ACTION ResetLockDepalletizing_2_action:
LockDepalletizing := FALSE;
END_ACTION

ACTION Check_StackIn__entry:
Delay.IN:=FALSE;
Delay();
END_ACTION

ACTION Check_StackIn__action:
Delay.IN:=ST08_404_B52_2.BitInToCheck;
Delay.PT:=T#3500ms;
Delay();
END_ACTION

ACTION VakuumOff_action:
ST08_403_Y50_6.MoveInit := TRUE;
ST08_403_Y50_7.MoveInit := TRUE;
END_ACTION

ACTION VakuumOff__action:
ST08_403_Y50_6.MoveInit := TRUE;
ST08_403_Y50_7.MoveInit := TRUE;
END_ACTION

ACTION SetLockDepalletizing_3_action:
LockDepalletizing := TRUE;
END_ACTION

ACTION CheckFixerPal_1_entry:
ProcessMessage02:='2IM1';(*'Abstapler wartet auf Aufstapler*)
END_ACTION

ACTION CheckFixerPal_1_exit:
ProcessMessage02:='';
END_ACTION

ACTION UnLocking_Trays_1__action:
ST08_405_Y53_4.MoveWork:=TRUE;
END_ACTION

ACTION Depallatizing_Unlock8_action:
LockDepalletizing := FALSE;
END_ACTION

ACTION Wait_Tray_entry:
Delay.IN:=FALSE;
Delay();
Timeout();
ProcessMessage01:='';
END_ACTION

ACTION Wait_Tray_action:
Delay(IN:=	NOT ST08_402_B51_2.BitInToCheck AND
     		ST08_404_B52_2.BitInToCheck
    ,PT:=T#300ms);

(*Damit der Aufstapler weitermachen kann, wenn kein Blister mehr kommt*)
Timeout(IN:=	NOT Delay.Q AND ST08_Palletizing.State=STATE_RUN, PT:=T#15s);
ProcessMessage01:='1IM16';(*ST. 8 warte aut Tray in HV vor Schleuse einlauf*)
END_ACTION

ACTION Locking_Trays___entry:
Timeout(IN:=FALSE);
END_ACTION

ACTION Locking_Trays___action:
ST08_405_Y53_4.MoveInit:=TRUE;
END_ACTION

ACTION Locking_Trays___exit:
gNewStackIn:=FALSE;
END_ACTION

ACTION Check_Blister__entry:
Delay(IN:=FALSE);
Timeout(IN:=FALSE);
END_ACTION

ACTION Check_Blister__action:
Delay(IN:=ST08_404_B52_3.BitInToCheck ,PT:=T#3000ms);
END_ACTION

ACTION Msg_SpecialMenu_entry:
MessageHandler.ClearMessageLines(sVisu:=Visu.Message);

MsgID:='PM200';
MsgString:='Blister falsche Lage in Blistereinlauf';
MsgString:=CONCAT(MsgString,'$R$N');
MsgString:=CONCAT(MsgString,'Lage korrigieren und weiter mit OK');
END_ACTION

ACTION Msg_SpecialMenu_action:
MessageHandler.Msg.ID:=MsgID;
MessageHandler.Msg.Name:='St8_Stop';
MessageHandler.Msg.Text:=MsgString;
MessageHandler.Msg.Color:=Color.red;
MessageHandler.Msg.Station:=5;
MessageHandler.MsgButton1Text:='continue';

MessageHandler(
	Prio:=2, 							(*1=highest, .. , 4=lowest*)
	Btn1Addr:=ADR(MsgOk),			(*Address of Button1 , if Zero then Button is unvisible*)
	Btn2Addr:=0,	(*Address of Button2 , if Zero then Button is unvisible*)
	sVisu:=Visu.Message);

MessageHandler.DisableMultiSelect(sVisu:=Visu.Message);
END_ACTION

ACTION Msg_SpecialMenu_exit:
MsgOk:=FALSE;
MsgCancel:=FALSE;
MessageHandler.ClearMessageLines(sVisu:=Visu.Message);
END_ACTION

ACTION Wait_DoorClose12_entry:
ProcessMessage01:='';
END_ACTION

ACTION Wait_DoorClose12_action:
ProcessMessage01:='1IM17';(*St. 8 warte Türe 2 Einlauf geschlossen*)
END_ACTION

ACTION Wait_DoorClose12_exit:
ProcessMessage01:='';
END_ACTION

ACTION Belt_on_action:
ConveyorOn:=TRUE;
END_ACTION

ACTION VRZ_open_action:
ST08_402_Y50_4.MoveWork:=TRUE;
END_ACTION

ACTION schieben_work_action:
ST08_402_Y52_7.MoveWork:=TRUE;
END_ACTION

ACTION Blister_Out_entry:
ProcessMessage01:='';
END_ACTION

ACTION Blister_Out_action:
ProcessMessage01:='1IM18';(*St. 8 warte aut Tray in Schleuse einlauf*)
END_ACTION

ACTION Blister_Out_exit:
gNewStackIn:=TRUE;
gRequestNewStack:=FALSE;
END_ACTION

ACTION VRZ_close_action:
ST08_402_Y50_4.MoveInit:=TRUE;
END_ACTION

ACTION schieben_init_action:
ST08_402_Y52_7.MoveInit:=TRUE;
END_ACTION

ACTION Belt_off_action:
ConveyorOn:=FALSE;
END_ACTION

ACTION Settling_time__entry:
Delay.IN:=FALSE;
Delay();
END_ACTION

ACTION Settling_time__action:
Delay.IN:=TRUE;
Delay.PT:=t#1000ms;
Delay();
END_ACTION

ACTION Check_StackIn___entry:
gRequestNewStack:=TRUE;
END_ACTION

ACTION Wait_DoorClose4_entry:
ProcessMessage01:='';
END_ACTION

ACTION Wait_DoorClose4_action:
ProcessMessage01:='1IM19';(*St.8 warte Türe 1 einlauf geschlossen*)
END_ACTION

ACTION Wait_DoorClose4_exit:
ProcessMessage01:='';
END_ACTION

ACTION Door_open_13_action:
ST08_405_Y51_0.MoveWork:=TRUE;
END_ACTION

ACTION VRZ_open_13_action:
ST08_404_Y51_6.MoveWork:=TRUE;
END_ACTION

ACTION Belt_on_13_action:
ConveyorOn:=TRUE;
END_ACTION

ACTION Check_TrayIn___entry:
ProcessMessage01:='';
END_ACTION

ACTION Check_TrayIn___action:
ProcessMessage01:='1IM20';(*St.4 warte auf Tray in Reinigungsposition*)
END_ACTION

ACTION Check_TrayIn___exit:
ProcessMessage01:='';
END_ACTION

ACTION VRZ_close_12_action:
ST08_404_Y51_6.MoveInit:=TRUE;
END_ACTION

ACTION Door_CLOSE_12_action:
ST08_405_Y51_0.MoveInit:=TRUE;
END_ACTION

ACTION Wait_DoorClose_5_entry:
ProcessMessage01:='';
END_ACTION

ACTION Wait_DoorClose_5_action:
ProcessMessage01:='1IM21';(*St.8 warte Türe 2 einlauf geschlossen*)
END_ACTION

ACTION Wait_DoorClose_5_exit:
ProcessMessage01:='';
END_ACTION

ACTION Belt_off_12_action:
ConveyorOn:=FALSE;
END_ACTION

ACTION ResultOk_action:
Result:=RESULT_OK;
END_ACTION

ACTION eWaitLastTray_entry:
ProcessMessage02:='EMPTY';
END_ACTION

ACTION eWaitLastTray_action:
ProcessMessage02:='2IM7';(*Aufstapler leerfahren*)
END_ACTION

ACTION eWaitLastTray_exit:
ProcessMessage02:='2IM8';(*Halb vollen Blister rausfahren*)
END_ACTION

ACTION eSetLockDepalletizing_2_action:
LockDepalletizing := TRUE;
END_ACTION

ACTION eM_Abstapeln_mitte_entry:
ST08_180_M1.MoveAbs:=TRUE;
ST08_180_M1.Vorgabe_Pos_Abs:=TD.PosAbstapeln[2].Pos;	(*1=unten, 2= mitte, 3=oben, 4=frei*)
END_ACTION

ACTION eLifter_Short_up_action:
ST08_404_Y53_0.MoveWork:=TRUE;
END_ACTION

ACTION eLifter_Long_down_action:
ST08_404_Y53_2.MoveInit:=TRUE;
END_ACTION

ACTION eVakuumOn_action:
ST08_403_Y50_6.MoveWork := TRUE;
ST08_403_Y50_7.MoveWork := TRUE;
END_ACTION

ACTION eCheckFixerPal__entry:
ProcessMessage02:='2IM1';(*'Abstapler wartet auf Aufstapler*)
END_ACTION

ACTION eCheckFixerPal__exit:
ProcessMessage02:='';
END_ACTION

ACTION eUnLocking_Trays__action:
ST08_405_Y53_4.MoveWork:=TRUE;
END_ACTION

ACTION eM_Abstapeln_unten___entry:
ST08_180_M1.MoveAbs:=TRUE;
ST08_180_M1.Vorgabe_Pos_Abs:=TD.PosAbstapeln[1].Pos;	(*1=unten, 2= mitte, 3=oben, 4=frei*)
END_ACTION

ACTION eLifter_Short_Down__action:
ST08_404_Y53_0.MoveInit:=TRUE;
END_ACTION

ACTION eResetLockDepalletizing_3_action:
LockDepalletizing := FALSE;
END_ACTION

ACTION eVakuumOff_action:
ST08_403_Y50_6.MoveInit := TRUE;
ST08_403_Y50_7.MoveInit := TRUE;
END_ACTION

ACTION eMsgEndRunEmpty_entry:
MessageHandler.ClearMessageLines(sVisu:=Visu.Message);
MsgOk:=FALSE;
ProcessMessage02:='EMPTY';
END_ACTION

ACTION eMsgEndRunEmpty_action:
MessageHandler.Msg.ID:='PM21';
MessageHandler.Msg.Name:='Maschine ist leergefahren';
MessageHandler.Msg.Text:= 'Maschine ist leergefahren';
MessageHandler.Msg.Color:=	Color.yellow ;
MessageHandler.Msg.Station:=1;

MessageHandler(
	Prio:=2, 					(*1=highest, .. , 4=lowest*)
	Btn1Addr:=ADR(MsgOk),		(*Address of Button1 , if Zero then Button is unvisible*)
	Btn2Addr:=0,				(*Address of Button2 , if Zero then Button is unvisible*)
	sVisu:=Visu.Message);

IF ModeSelect.Mode<=MODE_MANUAL THEN
	MsgOk:=TRUE;
END_IF
END_ACTION

ACTION eMsgEndRunEmpty_exit:
MsgOk:=FALSE;
ModeSelect.AskForManual:=TRUE;
gRunEmpty:=FALSE;
END_ACTION

ACTION SeqEnd_action:
SFCTime:=TIME_TO_DINT(TIME()-SFCTimeStart);
State:=STATE_WAIT;
END_ACTION

TRANSITION StateOk:
ST08_405_Y51_0.State=STATE_OK
END_TRANSITION

TRANSITION OK:
ST00_226_S2.BitInToCheck=FALSE
END_TRANSITION

TRANSITION with_Motor:
MP.ST08.StapelMotor
END_TRANSITION

TRANSITION MotorOn:
ST08_180_M1.On
END_TRANSITION

TRANSITION busy:
ST08_180_M1.Busy
END_TRANSITION

TRANSITION Done:
ST08_180_M1.Done
END_TRANSITION

TRANSITION StateOk:
ST08_404_Y53_2.State=STATE_OK
END_TRANSITION

TRANSITION StateOk:
ST08_404_Y53_0.State=STATE_OK
END_TRANSITION

TRANSITION OLD_:
NOT gNewStackIn AND
ST08_405_Y53_4.InitPosition
END_TRANSITION

TRANSITION free:
NOT ST08_Palletizing.LockPalletizing
END_TRANSITION

TRANSITION CheckClosePal:
ST08_408_B56_1.ValveSensor AND	 	(* Rückhaltezylinder links Auslauf STN8 GST *)
ST08_408_B56_3.ValveSensor 			(* Rückhaltezylinder rechts Auslauf STN8 GST *)
END_TRANSITION

TRANSITION StateOk:
ST08_405_Y53_4.State=STATE_OK
END_TRANSITION

TRANSITION with_Motor:
MP.ST08.StapelMotor
END_TRANSITION

TRANSITION on:
ST08_180_M1.on
END_TRANSITION

TRANSITION busy:
ST08_180_M1.Busy
END_TRANSITION

TRANSITION Done:
ST08_180_M1.Done
END_TRANSITION

TRANSITION StateOk:
ST08_404_Y53_0.State=STATE_OK
END_TRANSITION

TRANSITION StateOk:
ST08_405_Y53_4.State=STATE_OK
END_TRANSITION

TRANSITION with_Motor:
MP.ST08.StapelMotor
END_TRANSITION

TRANSITION VacuumOn:
ST08_403_Y50_6.State=STATE_OK AND
ST08_403_Y50_7.State=STATE_OK
END_TRANSITION

TRANSITION on:
ST08_180_M1.on
END_TRANSITION

TRANSITION busy:
ST08_180_M1.Busy
END_TRANSITION

TRANSITION Done:
ST08_180_M1.Done
END_TRANSITION

TRANSITION StateOk:
ST08_404_Y53_0.State=STATE_OK
END_TRANSITION

TRANSITION OK:
ST08_404_B52_2.BitInToCheck=FALSE OR Delay.Q
END_TRANSITION

TRANSITION VacuumOff:
ST08_403_Y50_6.State=STATE_OK AND
ST08_403_Y50_7.State=STATE_OK
END_TRANSITION

TRANSITION OK:
  DelayOut.Q
END_TRANSITION

TRANSITION Empty_:
Delay.Q
END_TRANSITION

TRANSITION free:
NOT ST08_Palletizing.LockPalletizing
END_TRANSITION

TRANSITION AutoStop:
		ModeSelect.Mode=MODE_AUTO_STOP
OR	ModeSelect.Mode=MODE_STEP_STOP
END_TRANSITION

TRANSITION with_Motor:
MP.ST08.StapelMotor
END_TRANSITION

TRANSITION MotorOn:
ST08_180_M1.On
END_TRANSITION

TRANSITION busy:
ST08_180_M1.Busy
END_TRANSITION

TRANSITION Done:
ST08_180_M1.Done
END_TRANSITION

TRANSITION StateOk:
ST08_404_Y53_0.State=STATE_OK
END_TRANSITION

TRANSITION StateOk:
ST08_404_Y53_2.State=STATE_OK
END_TRANSITION

TRANSITION VakuumOn:
ST08_403_Y50_6.State=STATE_OK AND
ST08_403_Y50_7.State=STATE_OK
END_TRANSITION

TRANSITION CheckClosePal:
ST08_408_B56_1.ValveSensor AND	 	(* Rückhaltezylinder links Auslauf STN8 GST *)
ST08_408_B56_3.ValveSensor 			(* Rückhaltezylinder rechts Auslauf STN8 GST *)
END_TRANSITION

TRANSITION StateOk:
ST08_405_Y53_4.State=STATE_OK
END_TRANSITION

TRANSITION with_Motor:
MP.ST08.StapelMotor
END_TRANSITION

TRANSITION MotorOn:
ST08_180_M1.On
END_TRANSITION

TRANSITION busy:
ST08_180_M1.Busy
END_TRANSITION

TRANSITION Done:
ST08_180_M1.Done
END_TRANSITION

TRANSITION StateOk:
ST08_404_Y53_2.State=STATE_OK
END_TRANSITION

TRANSITION StateOk:
ST08_405_Y53_4.State=STATE_OK
END_TRANSITION

TRANSITION with_Motor:
MP.ST08.StapelMotor
END_TRANSITION

TRANSITION MotorOn:
ST08_180_M1.On
END_TRANSITION

TRANSITION busy:
ST08_180_M1.Busy
END_TRANSITION

TRANSITION Done:
ST08_180_M1.Done
END_TRANSITION

TRANSITION StateOk:
ST08_404_Y53_0.State=STATE_OK
END_TRANSITION

TRANSITION In_:
ST08_404_B52_2.BitInToCheck=FALSE
END_TRANSITION

TRANSITION VakuumOff:
ST08_403_Y50_6.State=STATE_OK AND
ST08_403_Y50_7.State=STATE_OK
END_TRANSITION

TRANSITION Empty__:
Delay.Q
END_TRANSITION

TRANSITION VakuumOff:
ST08_403_Y50_6.State=STATE_OK AND
ST08_403_Y50_7.State=STATE_OK
END_TRANSITION

TRANSITION Trans90:
NOT ST08_Palletizing.LockPalletizing
END_TRANSITION

TRANSITION CheckClosePal:
ST08_408_B56_1.ValveSensor AND	 	(* Rückhaltezylinder links Auslauf STN8 GST *)
ST08_408_B56_3.ValveSensor 			(* Rückhaltezylinder rechts Auslauf STN8 GST *)
END_TRANSITION

TRANSITION StateOk:
ST08_405_Y53_4.State=STATE_OK
END_TRANSITION

TRANSITION AutoStop:
		ModeSelect.Mode=MODE_AUTO_STOP
OR	ModeSelect.Mode=MODE_STEP_STOP
END_TRANSITION

TRANSITION StateOk:
ST08_405_Y53_4.State=STATE_OK
END_TRANSITION

TRANSITION OK:
ST08_404_B52_3.BitInToCheck=FALSE OR
MP.ST03.SGM_3621
END_TRANSITION

TRANSITION TimeOut:
Delay.Q
END_TRANSITION

TRANSITION MsgOk:
		ST08_404_B52_3.BitInToCheck=FALSE
OR	MsgOk
END_TRANSITION

TRANSITION OK:
ST00_226_S2.BitInToCheck=FALSE
END_TRANSITION

TRANSITION StateOk:
ST08_402_Y50_4.State=STATE_OK
END_TRANSITION

TRANSITION mit_schieben:
MP.ST08.Traystapel_schieben
END_TRANSITION

TRANSITION #StateOk:
ST08_402_Y52_7.State=STATE_OK
END_TRANSITION

TRANSITION WTOut:
ST08_404_B52_2.BitInToCheck=FALSE AND ST08_402_B51_2.BitInToCheck=TRUE
END_TRANSITION

TRANSITION StateOk:
ST08_402_Y50_4.State=STATE_OK
END_TRANSITION

TRANSITION mit_schieben:
MP.ST08.Traystapel_schieben
END_TRANSITION

TRANSITION StateOk:
ST08_402_Y52_7.State=STATE_OK
END_TRANSITION

TRANSITION OK:
ST08_402_B51_5.BitInToCheck
END_TRANSITION

TRANSITION IN__:
 ST08_404_B52_2.BitInToCheck=FALSE
END_TRANSITION

TRANSITION OK:
NOT ST00_226_S1.BitInToCheck AND
NOT ST00_229_S1.BitInToCheck
END_TRANSITION

TRANSITION StateOk:
ST08_405_Y51_0.State=STATE_OK AND
ST08_404_Y51_6.State=STATE_OK
END_TRANSITION

TRANSITION OK:
    ST08_406_B54_0.BitInToCheck=FALSE AND ST08_404_B52_2.BitInToCheck=TRUE
END_TRANSITION

TRANSITION StateOk:
ST08_404_Y51_6.State=STATE_OK AND
ST08_405_Y51_0.State=STATE_OK
END_TRANSITION

TRANSITION OK:
ST00_226_S2.BitInToCheck=FALSE
END_TRANSITION

TRANSITION wait:
ST08_Palletizing.WaitLastTray
END_TRANSITION

TRANSITION voll:
NOT ST08_404_B52_2.BitInToCheck 		(*Traystapel in Ablageposition Isokörper*)
END_TRANSITION

TRANSITION leer:
ST08_404_B52_2.BitInToCheck 		(*Traystapel in Ablageposition Isokörper*)
END_TRANSITION

TRANSITION free:
NOT ST08_Palletizing.LockPalletizing
END_TRANSITION

TRANSITION with_Motor:
MP.ST08.StapelMotor
END_TRANSITION

TRANSITION MotorOn:
ST08_180_M1.On
END_TRANSITION

TRANSITION busy:
ST08_180_M1.Busy
END_TRANSITION

TRANSITION Done:
ST08_180_M1.Done
END_TRANSITION

TRANSITION StateOk:
ST08_404_Y53_0.State=STATE_OK
END_TRANSITION

TRANSITION StateOk:
ST08_404_Y53_2.State=STATE_OK
END_TRANSITION

TRANSITION VakuumOn:
ST08_403_Y50_6.State=STATE_OK AND
ST08_403_Y50_7.State=STATE_OK
END_TRANSITION

TRANSITION CheckClosePal:
ST08_408_B56_1.ValveSensor AND	 	(* Rückhaltezylinder links Auslauf STN8 GST *)
ST08_408_B56_3.ValveSensor 			(* Rückhaltezylinder rechts Auslauf STN8 GST *)
END_TRANSITION

TRANSITION StateOk:
ST08_405_Y53_4.State=STATE_OK
END_TRANSITION

TRANSITION with_Motor:
MP.ST08.StapelMotor
END_TRANSITION

TRANSITION MotorOn:
ST08_180_M1.On
END_TRANSITION

TRANSITION busy:
ST08_180_M1.Busy
END_TRANSITION

TRANSITION Done:
ST08_180_M1.Done
END_TRANSITION

TRANSITION StateOk:
ST08_404_Y53_0.State=STATE_OK
END_TRANSITION

TRANSITION VakuumOff:
ST08_403_Y50_6.State=STATE_OK AND
ST08_403_Y50_7.State=STATE_OK
END_TRANSITION

TRANSITION wait:
ST08_Palletizing.State = STATE_WAIT
END_TRANSITION
END_PROGRAM

(* POU Stations/ST_00/ST00_SFCs/_SpecialModeSFCs/SpecialMode01, SFC *)
PROGRAM SpecialMode01 (*Feeding-Test: Pickup Part with Robot01 from Feeder and put it into NOK-Box *)
(* Date: 07.DEZ 2010    Author: Ext/g.baiz  *)

VAR_OUTPUT
	SFCCurrentPOU		: STRING:='SpecialMode01';
	SFCCurrentStep	: STRING:='';
	SFCTime					:	DINT;
  State   				:	DINT;
  Result  				:	DINT;
END_VAR
VAR_INPUT
	Start						:	BOOL;
END_VAR
VAR
	MsgOK				:	BOOL;
	MsgCancel		:	BOOL;
	SFCRun					:	BOOL;
	SFCTimeStart		:	TIME;
	(* Userdefinded area *)



END_VAR
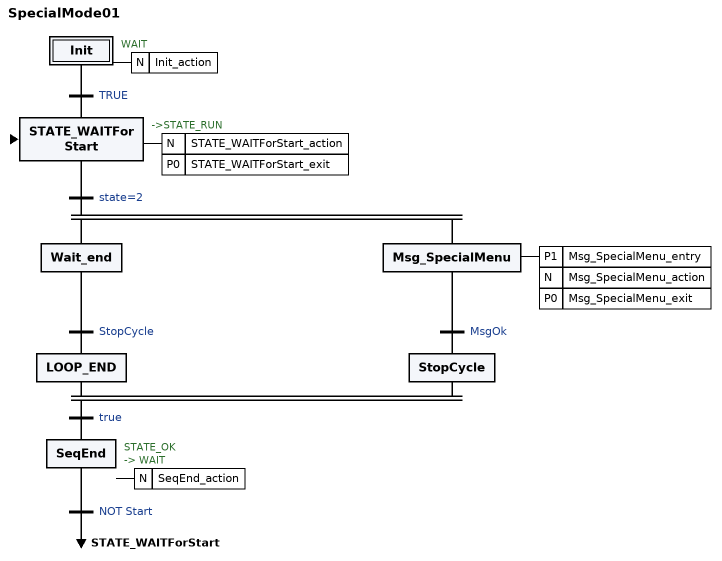
INITIAL_STEP Init: (* WAIT *)
	Init_action(N);
END_STEP
TRANSITION FROM Init TO STATE_WAITForStart := TRUE;
END_TRANSITION
STEP STATE_WAITForStart: (* ->STATE_RUN *)
	STATE_WAITForStart_action(N);
	STATE_WAITForStart_exit(P0);
END_STEP
TRANSITION FROM STATE_WAITForStart TO (Wait_end, Msg_SpecialMenu) := state=2;
END_TRANSITION
STEP Wait_end:
END_STEP
TRANSITION FROM Wait_end TO LOOP_END := StopCycle;
END_TRANSITION
STEP LOOP_END:
END_STEP
STEP Msg_SpecialMenu:
	Msg_SpecialMenu_entry(P1);
	Msg_SpecialMenu_action(N);
	Msg_SpecialMenu_exit(P0);
END_STEP
TRANSITION FROM Msg_SpecialMenu TO StopCycle := MsgOk;
END_TRANSITION
STEP StopCycle:
END_STEP
TRANSITION FROM (LOOP_END, StopCycle) TO SeqEnd := true;
END_TRANSITION
STEP SeqEnd: (* STATE_OK / -> WAIT *)
	SeqEnd_action(N);
END_STEP
TRANSITION FROM SeqEnd TO STATE_WAITForStart := NOT Start;
END_TRANSITION

ACTION Init_action:
Start:=FALSE;
State:=STATE_WAIT;
END_ACTION

ACTION STATE_WAITForStart_action:
IF 	Start THEN
	State:=STATE_RUN;
	Result:=RESULT_NON;
	SFCTimeStart:=TIME();
END_IF
END_ACTION

ACTION STATE_WAITForStart_exit:
StopCycle:=FALSE;
END_ACTION

ACTION Msg_SpecialMenu_entry:
MessageHandler.ClearMessageLines(sVisu:=Visu.Message);
StopCycle:=FALSE;
END_ACTION

ACTION Msg_SpecialMenu_action:
MessageHandler.Msg.ID:='PM50';
MessageHandler.Msg.Name:='SP1_Stop';
MessageHandler.Msg.Text:='Teilablauf beenden mit <OK>';
MessageHandler.Msg.Color:=Color.blue;
MessageHandler.Msg.Station:=0;


MessageHandler(
	Prio:=2, 									(*1=highest, .. , 4=lowest*)
	Btn1Addr:=ADR(MsgOk),			(*Address of Button1 , if Zero then Button is unvisible*)
	Btn2Addr:=0,	(*Address of Button2 , if Zero then Button is unvisible*)
	sVisu:=Visu.Message);

MessageHandler.DisableMultiSelect(sVisu:=Visu.Message);
END_ACTION

ACTION Msg_SpecialMenu_exit:
MsgOk:=FALSE;
MsgCancel:=FALSE;
StopCycle:=TRUE;
END_ACTION

ACTION SeqEnd_action:
IF 	State=STATE_RUN THEN
	SFCTime:=TIME_TO_DINT(TIME()-SFCTimeStart);
	State:=STATE_OK;
END_IF


IF 	NOT Start THEN
	State:=STATE_WAIT;
END_IF
END_ACTION
END_PROGRAM

(* POU Stations/ST_08_Palettierer/ST_08_SFCs/ST08_Palletizing, SFC *)
PROGRAM ST08_Palletizing

VAR_OUTPUT
	SFCCurrentPOU			: STRING:='ST08_Palletizing';
	SFCCurrentStep			: STRING:='';
	FB_CurrentStepHistorie	: FB_CurrentStepHistorie;
	SFCTime					: DINT;
	State   				: StateObject	:= STATE_WAIT;
	Result  				: StateResult;
	MoveInStopper			: BOOL;
END_VAR
VAR_INPUT
	TestpartMoveOut		: BOOL;
	MoveOut				: BOOL;
	ConveyorOn			: BOOL;
	LastTray			: BOOL;			(*Leerfahren. Der letzte, halbvollen Blisters ist rausgefahren*)
END_VAR
VAR
	MsgOK				: BOOL;
	MsgCancel			: BOOL;
	SFCRun				: BOOL;
	SFCTimeStart		: TIME;
	Delay				: TON;
	Error				: ErrorStruct;
	(* Userdefinded area *)
	ExitPosRdy_T		: TON;
	BlisterStart		: BOOL;
	LockInlett			:BOOL;

	WaitLastTray		:BOOL;		(*Leerfahren. Startet das Rausfahren des halbvollen Blisters*)
	LockPalletizing		:BOOL;
END_VAR
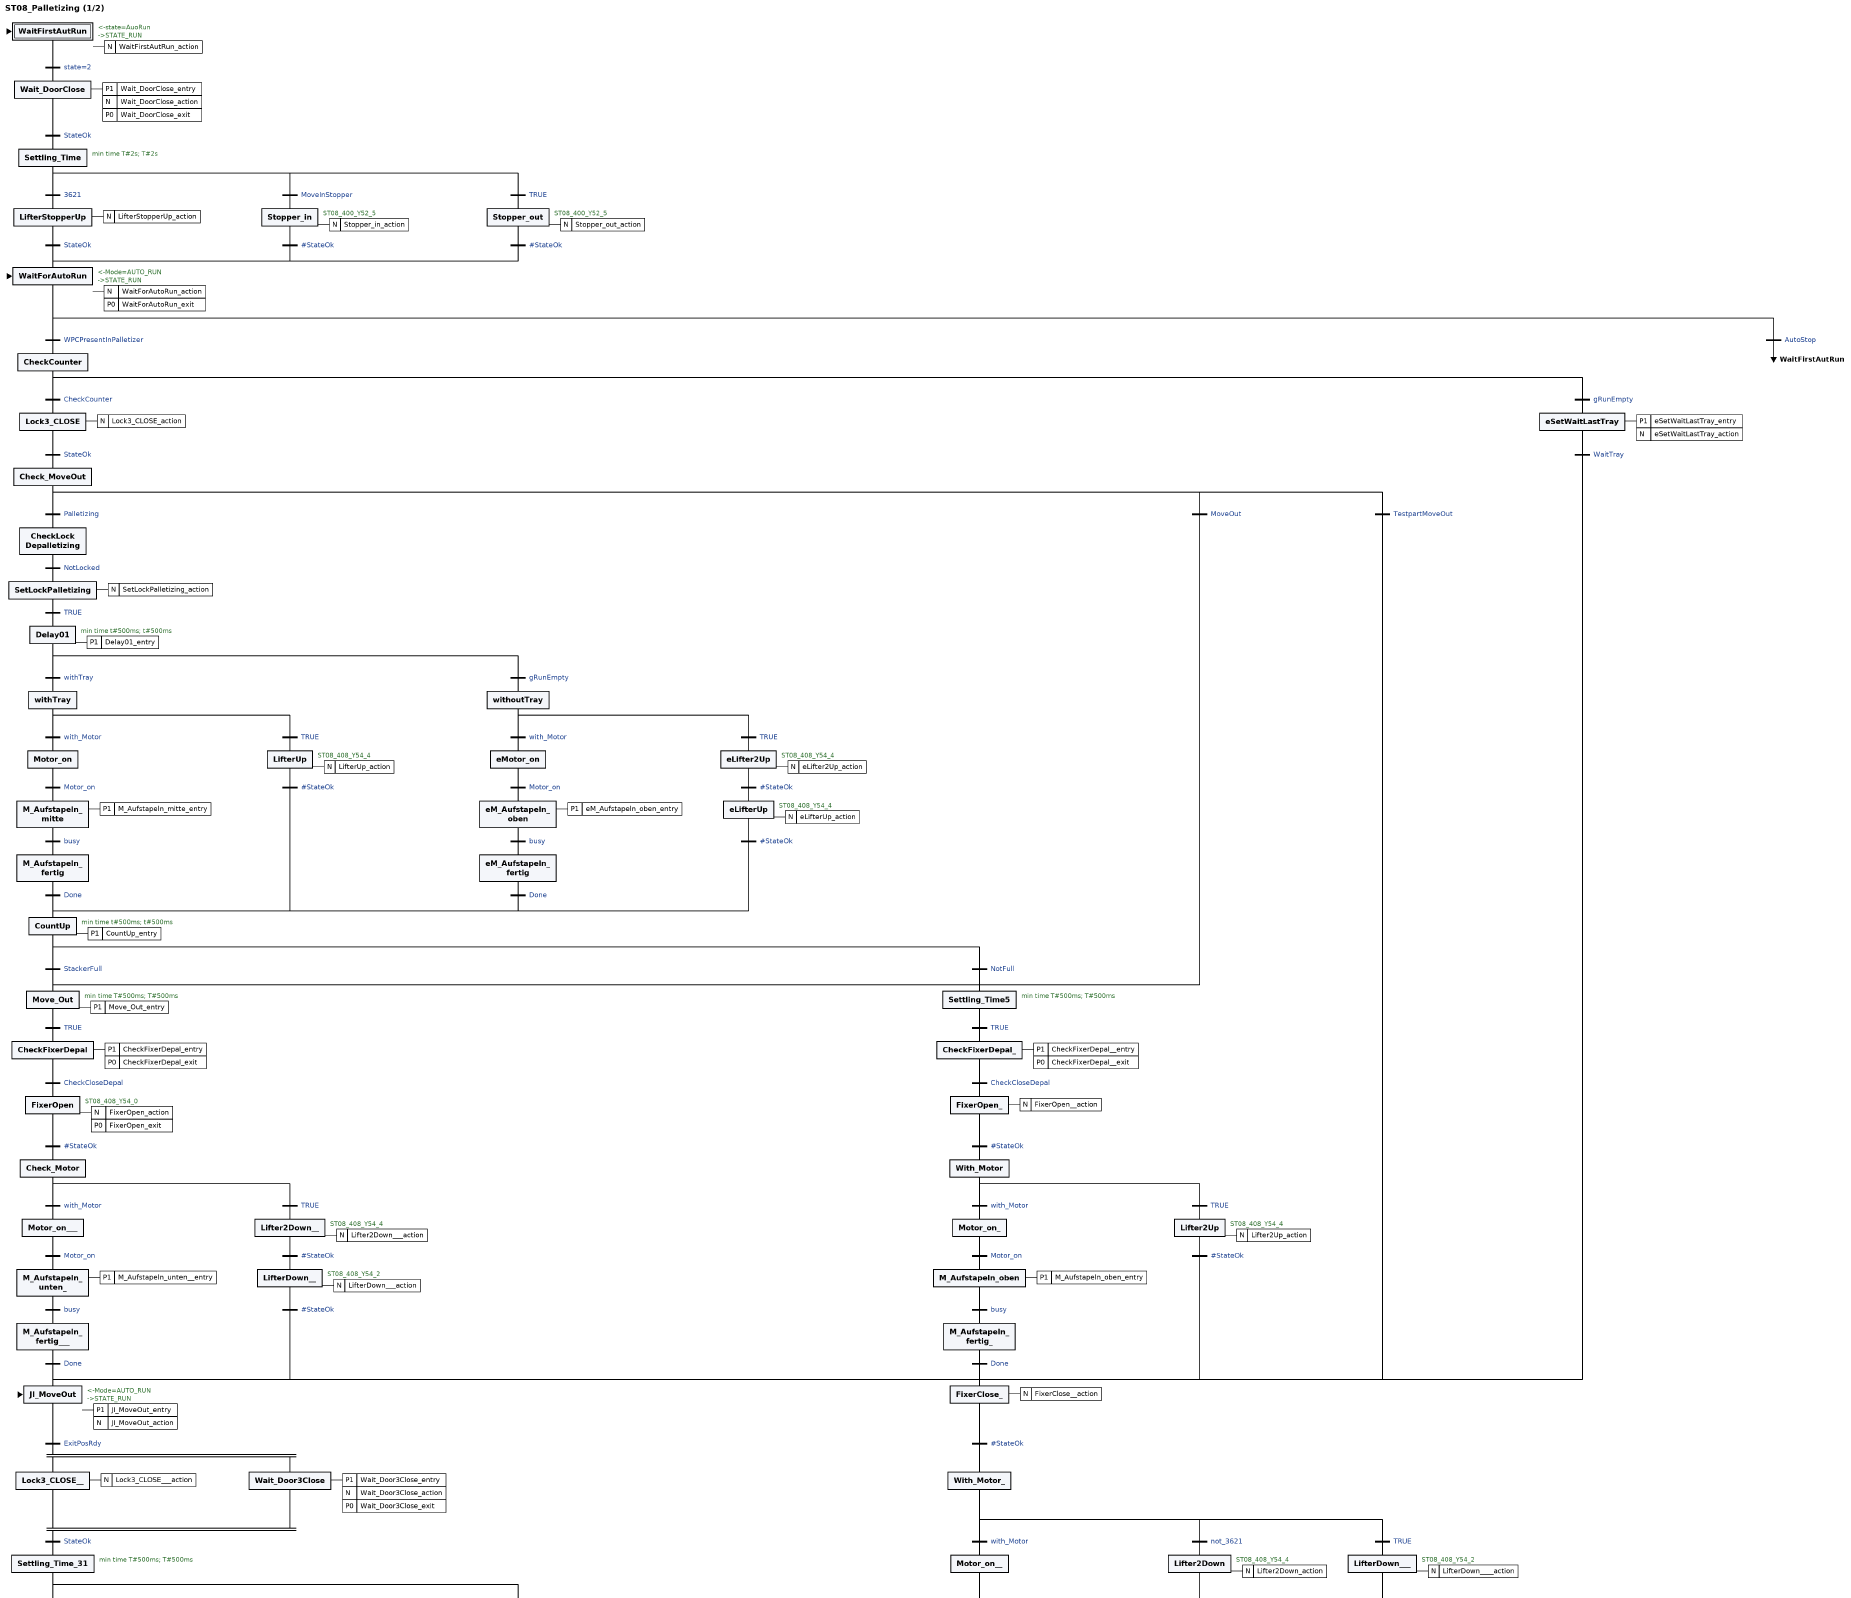
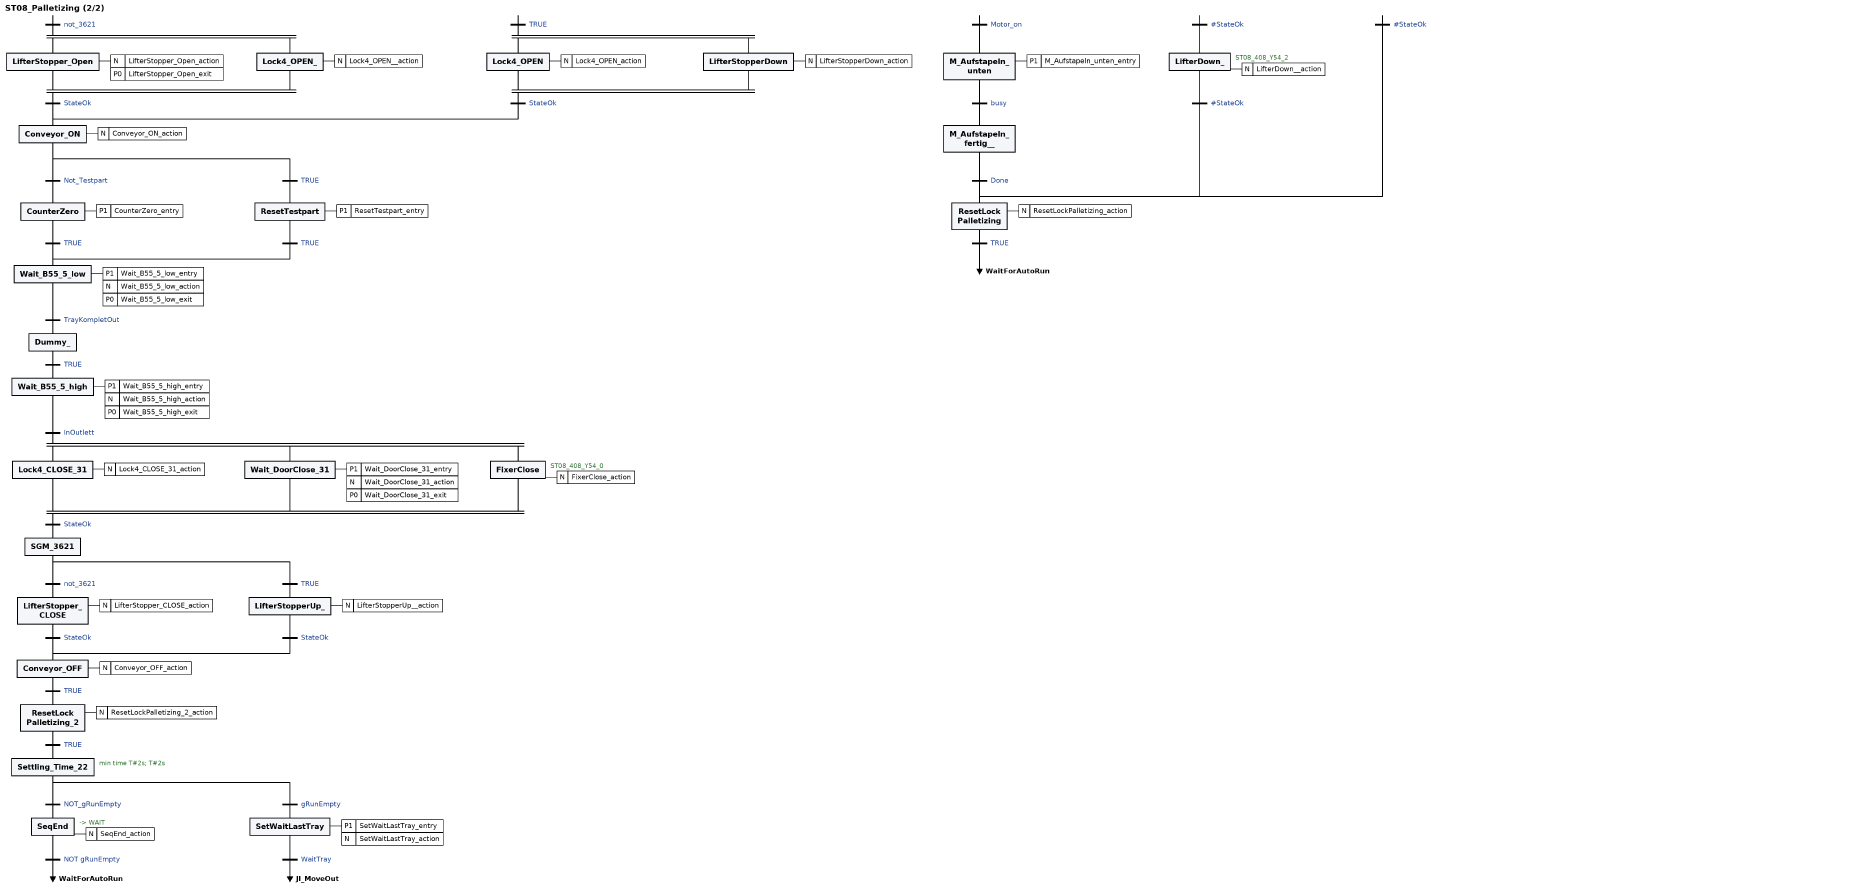
INITIAL_STEP WaitFirstAutRun: (* <-state=AuoRun / ->STATE_RUN *)
	WaitFirstAutRun_action(N);
END_STEP
TRANSITION FROM WaitFirstAutRun TO Wait_DoorClose := state=2;
END_TRANSITION
STEP Wait_DoorClose:
	Wait_DoorClose_entry(P1);
	Wait_DoorClose_action(N);
	Wait_DoorClose_exit(P0);
END_STEP
TRANSITION FROM Wait_DoorClose TO Settling_Time := StateOk;
END_TRANSITION
STEP Settling_Time: (* min time T#2s; T#2s *)
END_STEP
TRANSITION FROM Settling_Time TO LifterStopperUp := 3621;
END_TRANSITION
TRANSITION FROM Settling_Time TO Stopper_in := MoveInStopper;
END_TRANSITION
TRANSITION FROM Settling_Time TO Stopper_out := TRUE;
END_TRANSITION
STEP LifterStopperUp:
	LifterStopperUp_action(N);
END_STEP
TRANSITION FROM LifterStopperUp TO WaitForAutoRun := StateOk;
END_TRANSITION
STEP Stopper_in: (* ST08_400_Y52_5 *)
	Stopper_in_action(N);
END_STEP
TRANSITION FROM Stopper_in TO WaitForAutoRun := #StateOk;
END_TRANSITION
STEP Stopper_out: (* ST08_400_Y52_5 *)
	Stopper_out_action(N);
END_STEP
TRANSITION FROM Stopper_out TO WaitForAutoRun := #StateOk;
END_TRANSITION
STEP WaitForAutoRun: (* <-Mode=AUTO_RUN / ->STATE_RUN *)
	WaitForAutoRun_action(N);
	WaitForAutoRun_exit(P0);
END_STEP
TRANSITION FROM WaitForAutoRun TO CheckCounter := WPCPresentInPalletizer;
END_TRANSITION
TRANSITION FROM WaitForAutoRun TO WaitFirstAutRun := AutoStop;
END_TRANSITION
STEP CheckCounter:
END_STEP
TRANSITION FROM CheckCounter TO Lock3_CLOSE := CheckCounter;
END_TRANSITION
TRANSITION FROM CheckCounter TO eSetWaitLastTray := gRunEmpty;
END_TRANSITION
STEP eSetWaitLastTray:
	eSetWaitLastTray_entry(P1);
	eSetWaitLastTray_action(N);
END_STEP
TRANSITION FROM eSetWaitLastTray TO JI_MoveOut := WaitTray;
END_TRANSITION
STEP Lock3_CLOSE:
	Lock3_CLOSE_action(N);
END_STEP
TRANSITION FROM Lock3_CLOSE TO Check_MoveOut := StateOk;
END_TRANSITION
STEP Check_MoveOut:
END_STEP
TRANSITION FROM Check_MoveOut TO CheckLockDepalletizing := Palletizing;
END_TRANSITION
TRANSITION FROM Check_MoveOut TO Move_Out := MoveOut;
END_TRANSITION
TRANSITION FROM Check_MoveOut TO JI_MoveOut := TestpartMoveOut;
END_TRANSITION
STEP CheckLockDepalletizing:
END_STEP
TRANSITION FROM CheckLockDepalletizing TO SetLockPalletizing := NotLocked;
END_TRANSITION
STEP SetLockPalletizing:
	SetLockPalletizing_action(N);
END_STEP
TRANSITION FROM SetLockPalletizing TO Delay01 := TRUE;
END_TRANSITION
STEP Delay01: (* min time t#500ms; t#500ms *)
	Delay01_entry(P1);
END_STEP
TRANSITION FROM Delay01 TO withTray := withTray;
END_TRANSITION
TRANSITION FROM Delay01 TO withoutTray := gRunEmpty;
END_TRANSITION
STEP withTray:
END_STEP
TRANSITION FROM withTray TO Motor_on := with_Motor;
END_TRANSITION
TRANSITION FROM withTray TO LifterUp := TRUE;
END_TRANSITION
STEP Motor_on:
END_STEP
TRANSITION FROM Motor_on TO M_Aufstapeln_mitte := Motor_on;
END_TRANSITION
STEP M_Aufstapeln_mitte:
	M_Aufstapeln_mitte_entry(P1);
END_STEP
TRANSITION FROM M_Aufstapeln_mitte TO M_Aufstapeln_fertig := busy;
END_TRANSITION
STEP M_Aufstapeln_fertig:
END_STEP
TRANSITION FROM M_Aufstapeln_fertig TO CountUp := Done;
END_TRANSITION
STEP LifterUp: (* ST08_408_Y54_4 *)
	LifterUp_action(N);
END_STEP
TRANSITION FROM LifterUp TO CountUp := #StateOk;
END_TRANSITION
STEP withoutTray:
END_STEP
TRANSITION FROM withoutTray TO eMotor_on := with_Motor;
END_TRANSITION
TRANSITION FROM withoutTray TO eLifter2Up := TRUE;
END_TRANSITION
STEP eMotor_on:
END_STEP
TRANSITION FROM eMotor_on TO eM_Aufstapeln_oben := Motor_on;
END_TRANSITION
STEP eM_Aufstapeln_oben:
	eM_Aufstapeln_oben_entry(P1);
END_STEP
TRANSITION FROM eM_Aufstapeln_oben TO eM_Aufstapeln_fertig := busy;
END_TRANSITION
STEP eM_Aufstapeln_fertig:
END_STEP
TRANSITION FROM eM_Aufstapeln_fertig TO CountUp := Done;
END_TRANSITION
STEP eLifter2Up: (* ST08_408_Y54_4 *)
	eLifter2Up_action(N);
END_STEP
TRANSITION FROM eLifter2Up TO eLifterUp := #StateOk;
END_TRANSITION
STEP eLifterUp: (* ST08_408_Y54_4 *)
	eLifterUp_action(N);
END_STEP
TRANSITION FROM eLifterUp TO CountUp := #StateOk;
END_TRANSITION
STEP CountUp: (* min time t#500ms; t#500ms *)
	CountUp_entry(P1);
END_STEP
TRANSITION FROM CountUp TO Move_Out := StackerFull;
END_TRANSITION
TRANSITION FROM CountUp TO Settling_Time5 := NotFull;
END_TRANSITION
STEP Settling_Time5: (* min time T#500ms; T#500ms *)
END_STEP
TRANSITION FROM Settling_Time5 TO CheckFixerDepal_ := TRUE;
END_TRANSITION
STEP CheckFixerDepal_:
	CheckFixerDepal__entry(P1);
	CheckFixerDepal__exit(P0);
END_STEP
TRANSITION FROM CheckFixerDepal_ TO FixerOpen_ := CheckCloseDepal;
END_TRANSITION
STEP FixerOpen_:
	FixerOpen__action(N);
END_STEP
TRANSITION FROM FixerOpen_ TO With_Motor := #StateOk;
END_TRANSITION
STEP With_Motor:
END_STEP
TRANSITION FROM With_Motor TO Motor_on_ := with_Motor;
END_TRANSITION
TRANSITION FROM With_Motor TO Lifter2Up := TRUE;
END_TRANSITION
STEP Motor_on_:
END_STEP
TRANSITION FROM Motor_on_ TO M_Aufstapeln_oben := Motor_on;
END_TRANSITION
STEP M_Aufstapeln_oben:
	M_Aufstapeln_oben_entry(P1);
END_STEP
TRANSITION FROM M_Aufstapeln_oben TO M_Aufstapeln_fertig_ := busy;
END_TRANSITION
STEP M_Aufstapeln_fertig_:
END_STEP
TRANSITION FROM M_Aufstapeln_fertig_ TO FixerClose_ := Done;
END_TRANSITION
STEP Lifter2Up: (* ST08_408_Y54_4 *)
	Lifter2Up_action(N);
END_STEP
TRANSITION FROM Lifter2Up TO FixerClose_ := #StateOk;
END_TRANSITION
STEP FixerClose_:
	FixerClose__action(N);
END_STEP
TRANSITION FROM FixerClose_ TO With_Motor_ := #StateOk;
END_TRANSITION
STEP With_Motor_:
END_STEP
TRANSITION FROM With_Motor_ TO Motor_on__ := with_Motor;
END_TRANSITION
TRANSITION FROM With_Motor_ TO Lifter2Down := not_3621;
END_TRANSITION
TRANSITION FROM With_Motor_ TO LifterDown___ := TRUE;
END_TRANSITION
STEP Motor_on__:
END_STEP
TRANSITION FROM Motor_on__ TO M_Aufstapeln_unten := Motor_on;
END_TRANSITION
STEP M_Aufstapeln_unten:
	M_Aufstapeln_unten_entry(P1);
END_STEP
TRANSITION FROM M_Aufstapeln_unten TO M_Aufstapeln_fertig__ := busy;
END_TRANSITION
STEP M_Aufstapeln_fertig__:
END_STEP
TRANSITION FROM M_Aufstapeln_fertig__ TO ResetLockPalletizing := Done;
END_TRANSITION
STEP Lifter2Down: (* ST08_408_Y54_4 *)
	Lifter2Down_action(N);
END_STEP
TRANSITION FROM Lifter2Down TO LifterDown_ := #StateOk;
END_TRANSITION
STEP LifterDown_: (* ST08_408_Y54_2 *)
	LifterDown__action(N);
END_STEP
TRANSITION FROM LifterDown_ TO ResetLockPalletizing := #StateOk;
END_TRANSITION
STEP LifterDown___: (* ST08_408_Y54_2 *)
	LifterDown____action(N);
END_STEP
TRANSITION FROM LifterDown___ TO ResetLockPalletizing := #StateOk;
END_TRANSITION
STEP ResetLockPalletizing:
	ResetLockPalletizing_action(N);
END_STEP
TRANSITION FROM ResetLockPalletizing TO WaitForAutoRun := TRUE;
END_TRANSITION
STEP Move_Out: (* min time T#500ms; T#500ms *)
	Move_Out_entry(P1);
END_STEP
TRANSITION FROM Move_Out TO CheckFixerDepal := TRUE;
END_TRANSITION
STEP CheckFixerDepal:
	CheckFixerDepal_entry(P1);
	CheckFixerDepal_exit(P0);
END_STEP
TRANSITION FROM CheckFixerDepal TO FixerOpen := CheckCloseDepal;
END_TRANSITION
STEP FixerOpen: (* ST08_408_Y54_0 *)
	FixerOpen_action(N);
	FixerOpen_exit(P0);
END_STEP
TRANSITION FROM FixerOpen TO Check_Motor := #StateOk;
END_TRANSITION
STEP Check_Motor:
END_STEP
TRANSITION FROM Check_Motor TO Motor_on___ := with_Motor;
END_TRANSITION
TRANSITION FROM Check_Motor TO Lifter2Down__ := TRUE;
END_TRANSITION
STEP Motor_on___:
END_STEP
TRANSITION FROM Motor_on___ TO M_Aufstapeln_unten_ := Motor_on;
END_TRANSITION
STEP M_Aufstapeln_unten_:
	M_Aufstapeln_unten__entry(P1);
END_STEP
TRANSITION FROM M_Aufstapeln_unten_ TO M_Aufstapeln_fertig___ := busy;
END_TRANSITION
STEP M_Aufstapeln_fertig___:
END_STEP
TRANSITION FROM M_Aufstapeln_fertig___ TO JI_MoveOut := Done;
END_TRANSITION
STEP Lifter2Down__: (* ST08_408_Y54_4 *)
	Lifter2Down___action(N);
END_STEP
TRANSITION FROM Lifter2Down__ TO LifterDown__ := #StateOk;
END_TRANSITION
STEP LifterDown__: (* ST08_408_Y54_2 *)
	LifterDown___action(N);
END_STEP
TRANSITION FROM LifterDown__ TO JI_MoveOut := #StateOk;
END_TRANSITION
STEP JI_MoveOut: (* <-Mode=AUTO_RUN / ->STATE_RUN *)
	JI_MoveOut_entry(P1);
	JI_MoveOut_action(N);
END_STEP
TRANSITION FROM JI_MoveOut TO (Lock3_CLOSE__, Wait_Door3Close) := ExitPosRdy;
END_TRANSITION
STEP Lock3_CLOSE__:
	Lock3_CLOSE___action(N);
END_STEP
STEP Wait_Door3Close:
	Wait_Door3Close_entry(P1);
	Wait_Door3Close_action(N);
	Wait_Door3Close_exit(P0);
END_STEP
TRANSITION FROM (Lock3_CLOSE__, Wait_Door3Close) TO Settling_Time_31 := StateOk;
END_TRANSITION
STEP Settling_Time_31: (* min time T#500ms; T#500ms *)
END_STEP
TRANSITION FROM Settling_Time_31 TO (LifterStopper_Open, Lock4_OPEN_) := not_3621;
END_TRANSITION
TRANSITION FROM Settling_Time_31 TO (Lock4_OPEN, LifterStopperDown) := TRUE;
END_TRANSITION
STEP LifterStopper_Open:
	LifterStopper_Open_action(N);
	LifterStopper_Open_exit(P0);
END_STEP
STEP Lock4_OPEN_:
	Lock4_OPEN__action(N);
END_STEP
TRANSITION FROM (LifterStopper_Open, Lock4_OPEN_) TO Conveyor_ON := StateOk;
END_TRANSITION
STEP Lock4_OPEN:
	Lock4_OPEN_action(N);
END_STEP
STEP LifterStopperDown:
	LifterStopperDown_action(N);
END_STEP
TRANSITION FROM (Lock4_OPEN, LifterStopperDown) TO Conveyor_ON := StateOk;
END_TRANSITION
STEP Conveyor_ON:
	Conveyor_ON_action(N);
END_STEP
TRANSITION FROM Conveyor_ON TO CounterZero := Not_Testpart;
END_TRANSITION
TRANSITION FROM Conveyor_ON TO ResetTestpart := TRUE;
END_TRANSITION
STEP CounterZero:
	CounterZero_entry(P1);
END_STEP
TRANSITION FROM CounterZero TO Wait_B55_5_low := TRUE;
END_TRANSITION
STEP ResetTestpart:
	ResetTestpart_entry(P1);
END_STEP
TRANSITION FROM ResetTestpart TO Wait_B55_5_low := TRUE;
END_TRANSITION
STEP Wait_B55_5_low:
	Wait_B55_5_low_entry(P1);
	Wait_B55_5_low_action(N);
	Wait_B55_5_low_exit(P0);
END_STEP
TRANSITION FROM Wait_B55_5_low TO Dummy_ := TrayKompletOut;
END_TRANSITION
STEP Dummy_:
END_STEP
TRANSITION FROM Dummy_ TO Wait_B55_5_high := TRUE;
END_TRANSITION
STEP Wait_B55_5_high:
	Wait_B55_5_high_entry(P1);
	Wait_B55_5_high_action(N);
	Wait_B55_5_high_exit(P0);
END_STEP
TRANSITION FROM Wait_B55_5_high TO (Lock4_CLOSE_31, Wait_DoorClose_31, FixerClose) := InOutlett;
END_TRANSITION
STEP Lock4_CLOSE_31:
	Lock4_CLOSE_31_action(N);
END_STEP
STEP Wait_DoorClose_31:
	Wait_DoorClose_31_entry(P1);
	Wait_DoorClose_31_action(N);
	Wait_DoorClose_31_exit(P0);
END_STEP
STEP FixerClose: (* ST08_408_Y54_0 *)
	FixerClose_action(N);
END_STEP
TRANSITION FROM (Lock4_CLOSE_31, Wait_DoorClose_31, FixerClose) TO SGM_3621 := StateOk;
END_TRANSITION
STEP SGM_3621:
END_STEP
TRANSITION FROM SGM_3621 TO LifterStopper_CLOSE := not_3621;
END_TRANSITION
TRANSITION FROM SGM_3621 TO LifterStopperUp_ := TRUE;
END_TRANSITION
STEP LifterStopper_CLOSE:
	LifterStopper_CLOSE_action(N);
END_STEP
TRANSITION FROM LifterStopper_CLOSE TO Conveyor_OFF := StateOk;
END_TRANSITION
STEP LifterStopperUp_:
	LifterStopperUp__action(N);
END_STEP
TRANSITION FROM LifterStopperUp_ TO Conveyor_OFF := StateOk;
END_TRANSITION
STEP Conveyor_OFF:
	Conveyor_OFF_action(N);
END_STEP
TRANSITION FROM Conveyor_OFF TO ResetLockPalletizing_2 := TRUE;
END_TRANSITION
STEP ResetLockPalletizing_2:
	ResetLockPalletizing_2_action(N);
END_STEP
TRANSITION FROM ResetLockPalletizing_2 TO Settling_Time_22 := TRUE;
END_TRANSITION
STEP Settling_Time_22: (* min time T#2s; T#2s *)
END_STEP
TRANSITION FROM Settling_Time_22 TO SeqEnd := NOT_gRunEmpty;
END_TRANSITION
TRANSITION FROM Settling_Time_22 TO SetWaitLastTray := gRunEmpty;
END_TRANSITION
STEP SetWaitLastTray:
	SetWaitLastTray_entry(P1);
	SetWaitLastTray_action(N);
END_STEP
TRANSITION FROM SetWaitLastTray TO JI_MoveOut := WaitTray;
END_TRANSITION
STEP SeqEnd: (* -> WAIT *)
	SeqEnd_action(N);
END_STEP
TRANSITION FROM SeqEnd TO WaitForAutoRun := NOT gRunEmpty;
END_TRANSITION

ACTION WaitFirstAutRun_action:
IF 	ModeSelect.Mode=MODE_AUTO_RUN OR
	ModeSelect.Mode=MODE_STEP_RUN OR
	SpecialMode01.State=State_Run OR
 	SpecialMode06.State=State_Run THEN
	State:=STATE_RUN;
	Result:=RESULT_NON;
ELSE
	State:=STATE_WAIT;
END_IF
IF 	ModeSelect.Mode <> MODE_HOME_POS_RUN THEN
	ConveyorOn:=FALSE;
END_IF

MsgOK:=FALSE;
MsgCancel:=FALSE;
SFCRun:=FALSE;
BlisterStart:=FALSE;
LockInlett:=FALSE;
LockPalletizing:=FALSE;
MoveInStopper:=FALSE;
LastTray:=FALSE;
WaitLastTray:=FALSE;
END_ACTION

ACTION Wait_DoorClose_entry:
ProcessMessage01:='';
END_ACTION

ACTION Wait_DoorClose_action:
ProcessMessage01:='1IM8';(*St.8 warte Türe 4 auslauf geschlossen*)
ST08_407_Y51_4.MoveInit:=TRUE;
END_ACTION

ACTION Wait_DoorClose_exit:
ProcessMessage01:='';
END_ACTION

ACTION LifterStopperUp_action:
ST08_408_Y54_4.MoveWork:=TRUE;
END_ACTION

ACTION Stopper_in_action:
ST08_400_Y52_5.MoveWork :=TRUE; (* einfahren Stopper links + rechts Traystapel Auslaufband einfahren *)
END_ACTION

ACTION Stopper_out_action:
ST08_400_Y52_5.MoveInit :=TRUE; (* ausfahren Stopper links + rechts Traystapel Auslaufband einfahren *)
END_ACTION

ACTION WaitForAutoRun_action:
State:=STATE_WAIT;
LockInlett:=FALSE;
END_ACTION

ACTION WaitForAutoRun_exit:
State:=STATE_RUN;
Result:=RESULT_NON;
SFCTimeStart:=TIME();
END_ACTION

ACTION eSetWaitLastTray_entry:
LockInlett:=FALSE;
END_ACTION

ACTION eSetWaitLastTray_action:
WaitLastTray:=TRUE; (*damit wird im ST08_Process der halbvolle Blister ausgeschleust*)
END_ACTION

ACTION Lock3_CLOSE_action:
ST08_406_Y51_2.MoveInit:=TRUE;
END_ACTION

ACTION SetLockPalletizing_action:
LockPalletizing := TRUE;
END_ACTION

ACTION Delay01_entry:
LockInlett:=TRUE;
END_ACTION

ACTION M_Aufstapeln_mitte_entry:
ST08_185_M1.MoveAbs:=TRUE;
ST08_185_M1.Vorgabe_Pos_Abs:=TD.PosAufstapeln[2].Pos;	(*1=unten, 2= mitte, 3=oben, 4=frei*)
ST08_185_M1.Vorgabe_Velo:=1750;
END_ACTION

ACTION LifterUp_action:
ST08_408_Y54_2.MoveWork:=TRUE;
END_ACTION

ACTION eM_Aufstapeln_oben_entry:
ST08_185_M1.MoveAbs:=TRUE;
ST08_185_M1.Vorgabe_Pos_Abs:=TD.PosAufstapeln[3].Pos;	(*1=unten, 2= mitte, 3=oben, 4=frei*)
ST08_185_M1.Vorgabe_Velo:=1750;
END_ACTION

ACTION eLifter2Up_action:
ST08_408_Y54_4.MoveWork:=TRUE;
END_ACTION

ACTION eLifterUp_action:
ST08_408_Y54_2.MoveWork:=TRUE;
END_ACTION

ACTION CountUp_entry:
MP.ST08.NoOfBlisterInStackerOut:=MP.ST08.NoOfBlisterInStackerOut+1;
END_ACTION

ACTION CheckFixerDepal__entry:
ProcessMessage02:='2IM2';(*'Aufstapler wartet auf Abstapler*)
END_ACTION

ACTION CheckFixerDepal__exit:
ProcessMessage02:='';
END_ACTION

ACTION FixerOpen__action:
ST08_408_Y54_0.MoveWork:=TRUE;
END_ACTION

ACTION M_Aufstapeln_oben_entry:
ST08_185_M1.MoveAbs:=TRUE;
ST08_185_M1.Vorgabe_Pos_Abs:=TD.PosAufstapeln[3].Pos;	(*1=unten, 2= mitte, 3=oben, 4=frei*)
END_ACTION

ACTION Lifter2Up_action:
ST08_408_Y54_4.MoveWork:=TRUE;
END_ACTION

ACTION FixerClose__action:
ST08_408_Y54_0.MoveInit:=TRUE;
END_ACTION

ACTION M_Aufstapeln_unten_entry:
ST08_185_M1.MoveAbs:=TRUE;
ST08_185_M1.Vorgabe_Pos_Abs:=TD.PosAufstapeln[1].Pos;	(*1=unten, 2= mitte, 3=oben, 4=frei*)
END_ACTION

ACTION Lifter2Down_action:
ST08_408_Y54_4.MoveInit:=TRUE;
END_ACTION

ACTION LifterDown__action:
ST08_408_Y54_2.MoveInit:=TRUE;
END_ACTION

ACTION LifterDown____action:
ST08_408_Y54_2.MoveInit:=TRUE;
END_ACTION

ACTION ResetLockPalletizing_action:
LockPalletizing := FALSE;
END_ACTION

ACTION Move_Out_entry:
MoveOut:=TRUE;
END_ACTION

ACTION CheckFixerDepal_entry:
ProcessMessage02:='2IM2';(*'Aufstapler wartet auf Abstapler*)
END_ACTION

ACTION CheckFixerDepal_exit:
ProcessMessage02:='';
END_ACTION

ACTION FixerOpen_action:
ST08_408_Y54_0.MoveWork:=TRUE;
END_ACTION

ACTION FixerOpen_exit:
MP.ST03.WpcInStackFilled:=FALSE;
END_ACTION

ACTION M_Aufstapeln_unten__entry:
ST08_185_M1.MoveAbs:=TRUE;
ST08_185_M1.Vorgabe_Pos_Abs:=TD.PosAufstapeln[1].Pos;	(*1=unten, 2= mitte, 3=oben, 4=frei*)
END_ACTION

ACTION Lifter2Down___action:
ST08_408_Y54_4.MoveInit:=TRUE;
END_ACTION

ACTION LifterDown___action:
ST08_408_Y54_2.MoveInit:=TRUE;
END_ACTION

ACTION JI_MoveOut_entry:
ExitPosRdy_T(IN:=FALSE);
Delay.IN:=FALSE;
Delay();
END_ACTION

ACTION JI_MoveOut_action:
ExitPosRdy_T(IN:=
		(ModeSelect.Mode=MODE_AUTO_RUN	OR
		ModeSelect.Mode=MODE_STEP_RUN   OR
		ModeSelect.Mode=MODE_SPECIAL) AND
		ST08_409_B55_5.BitInToCheck , 	(* kein Stau im Auslauf *)
		PT:=T#2s);

Delay(IN:=TRUE,PT:=T#5s);

IF Delay.Q THEN
	MessageHandler.Msg.ID:='PM201';
	MessageHandler.Msg.Name:='St08 Stau im Auslauf';
	MessageHandler.Msg.Text:='Auslaufand voll!! Blister entnehmen!!';
	MessageHandler.Msg.Color:=Color.blue;
	MessageHandler.Msg.Station:=0;


	MessageHandler(
		Prio:=2, 		(*1=highest, .. , 4=lowest*)
		Btn1Addr:=0,	(*Address of Button1 , if Zero then Button is unvisible*)
		Btn2Addr:=0,	(*Address of Button2 , if Zero then Button is unvisible*)
		sVisu:=Visu.Message);


END_IF
END_ACTION

ACTION Lock3_CLOSE___action:
ST08_406_Y51_2.MoveInit:=TRUE;
END_ACTION

ACTION Wait_Door3Close_entry:
ProcessMessage01:='';
END_ACTION

ACTION Wait_Door3Close_action:
ProcessMessage01:='1IM11';(*St.8 warte Türe 3 auslauf geschlossen*)
END_ACTION

ACTION Wait_Door3Close_exit:
ProcessMessage01:='';
END_ACTION

ACTION LifterStopper_Open_action:
ST08_400_Y52_5.MoveWork :=TRUE;
END_ACTION

ACTION LifterStopper_Open_exit:
MoveInStopper:=TRUE;
END_ACTION

ACTION Lock4_OPEN__action:
ST08_407_Y51_4.MoveWork:=TRUE;
END_ACTION

ACTION Lock4_OPEN_action:
ST08_407_Y51_4.MoveWork:=TRUE;
END_ACTION

ACTION LifterStopperDown_action:
ST08_408_Y54_4.MoveInit:=TRUE;
END_ACTION

ACTION Conveyor_ON_action:
ConveyorOn:=TRUE;
END_ACTION

ACTION CounterZero_entry:
MP.ST08.NoOfBlisterInStackerOut:=0;
END_ACTION

ACTION ResetTestpart_entry:
TestpartMoveOut:=FALSE;
END_ACTION

ACTION Wait_B55_5_low_entry:
ProcessMessage01:='';
END_ACTION

ACTION Wait_B55_5_low_action:
ProcessMessage01:='1IM12';(*'St. 8 warte Tray ausgelaufen*)
END_ACTION

ACTION Wait_B55_5_low_exit:
ProcessMessage01:='';
END_ACTION

ACTION Wait_B55_5_high_entry:
ProcessMessage01:='';
END_ACTION

ACTION Wait_B55_5_high_action:
ProcessMessage01:='1IM13';(*St. 8 warte Tray auf Rollenbahn*)
END_ACTION

ACTION Wait_B55_5_high_exit:
MoveInStopper:=FALSE;
END_ACTION

ACTION Lock4_CLOSE_31_action:
ST08_407_Y51_4.MoveInit:=TRUE;
END_ACTION

ACTION Wait_DoorClose_31_entry:
ProcessMessage01:='';
END_ACTION

ACTION Wait_DoorClose_31_action:
ProcessMessage01:='1IM14';(*'St.8 warte Türe 4 auslauf geschlossen*)
END_ACTION

ACTION Wait_DoorClose_31_exit:
ProcessMessage01:='';
END_ACTION

ACTION FixerClose_action:
ST08_408_Y54_0.MoveInit:=TRUE;
END_ACTION

ACTION LifterStopper_CLOSE_action:
ST08_400_Y52_5.MoveInit:=TRUE;
END_ACTION

ACTION LifterStopperUp__action:
ST08_408_Y54_4.MoveWork:=TRUE;
END_ACTION

ACTION Conveyor_OFF_action:
ConveyorOn:=FALSE;
END_ACTION

ACTION ResetLockPalletizing_2_action:
LockPalletizing := FALSE;
END_ACTION

ACTION SetWaitLastTray_entry:
LockInlett:=FALSE;
END_ACTION

ACTION SetWaitLastTray_action:
WaitLastTray:=TRUE; (*damit wird im ST08_Process der halbvolle Blister ausgeschleust*)
END_ACTION

ACTION SeqEnd_action:
SFCTime:=TIME_TO_DINT(TIME()-SFCTimeStart);
State:=STATE_WAIT;
END_ACTION

TRANSITION StateOk:
ST08_407_Y51_4.State=STATE_OK AND
NOT ST00_227_S2.BitInToCheck AND
NOT ST00_230_S1.BitInToCheck
END_TRANSITION

TRANSITION 3621:
MP.ST03.SGM_3621
END_TRANSITION

TRANSITION StateOk:
ST08_408_Y54_4.State=STATE_OK

AND gTipImp
END_TRANSITION

TRANSITION #StateOk:
ST08_400_Y52_5.State=STATE_OK
AND gTipImp
END_TRANSITION

TRANSITION #StateOk:
ST08_400_Y52_5.State=STATE_OK
AND gTipImp
END_TRANSITION

TRANSITION WPCPresentInPalletizer:
(NOT ST08_407_B55_4.BitInToCheck OR
gRunEmpty)AND
gTipImp
END_TRANSITION

TRANSITION CheckCounter:
(gRunEmpty AND MP.ST08.NoOfBlisterInStackerOut >0) OR
NOT gRunEmpty
END_TRANSITION

TRANSITION gRunEmpty:
gRunEmpty AND MP.ST08.NoOfBlisterInStackerOut = 0
END_TRANSITION

TRANSITION WaitTray:
NOT ST08_407_B55_4.BitInToCheck AND	(* Tray in Aufstapelposition eingelaufen STN8 *)
LastTray AND	 (*damit wird im ST08_Process das ausschleusen des halbvollen Blisters bestätigt*)
gTipImp
END_TRANSITION

TRANSITION StateOk:
ST08_406_Y51_2.State=STATE_OK
END_TRANSITION

TRANSITION Palletizing:
NOT MoveOut AND
NOT TestpartMoveOut
END_TRANSITION

TRANSITION NotLocked:
NOT ST08_Depalletizing.LockDepalletizing
END_TRANSITION

TRANSITION withTray:
NOT ST08_407_B55_4.BitInToCheck (* Tray in Aufstapelposition eingelaufen STN8 *)
END_TRANSITION

TRANSITION with_Motor:
MP.ST08.StapelMotor
END_TRANSITION

TRANSITION Motor_on:
ST08_185_M1.On
END_TRANSITION

TRANSITION busy:
ST08_185_M1.Busy
END_TRANSITION

TRANSITION Done:
ST08_185_M1.Done
END_TRANSITION

TRANSITION #StateOk:
ST08_408_Y54_2.State=STATE_OK

AND gTipImp
END_TRANSITION

TRANSITION with_Motor:
MP.ST08.StapelMotor
END_TRANSITION

TRANSITION Motor_on:
ST08_185_M1.On
END_TRANSITION

TRANSITION busy:
ST08_185_M1.Busy
END_TRANSITION

TRANSITION Done:
ST08_185_M1.Done
END_TRANSITION

TRANSITION #StateOk:
ST08_408_Y54_4.State=STATE_OK

AND gTipImp
END_TRANSITION

TRANSITION #StateOk:
ST08_408_Y54_2.State=STATE_OK

AND gTipImp
END_TRANSITION

TRANSITION StackerFull:
MP.ST08.NoOfBlisterInStackerOut>=TD.NoOfPalletsPerStack OR
gRunEmpty
END_TRANSITION

TRANSITION NotFull:
TRUE
END_TRANSITION

TRANSITION CheckCloseDepal:
ST08_405_B53_3.ValveSensor AND	 	(* Rückhaltezylinder links Traystapel Isokörper GST *)
ST08_405_B53_5.ValveSensor 			(* Rückhaltezylinder rechts Traystapel Isokörper GST *)
END_TRANSITION

TRANSITION #StateOk:
ST08_408_Y54_0.State=STATE_OK

AND gTipImp
END_TRANSITION

TRANSITION with_Motor:
MP.ST08.StapelMotor
END_TRANSITION

TRANSITION Motor_on:
ST08_185_M1.On
END_TRANSITION

TRANSITION busy:
ST08_185_M1.Busy
END_TRANSITION

TRANSITION Done:
ST08_185_M1.Done AND
gTipImp
END_TRANSITION

TRANSITION #StateOk:
ST08_408_Y54_4.State=STATE_OK

AND gTipImp
END_TRANSITION

TRANSITION #StateOk:
ST08_408_Y54_0.State=STATE_OK

AND gTipImp
END_TRANSITION

TRANSITION with_Motor:
MP.ST08.StapelMotor
END_TRANSITION

TRANSITION Motor_on:
ST08_185_M1.On
END_TRANSITION

TRANSITION busy:
ST08_185_M1.Busy
END_TRANSITION

TRANSITION Done:
ST08_185_M1.Done AND
gTipImp
END_TRANSITION

TRANSITION not_3621:
NOT MP.ST03.SGM_3621
END_TRANSITION

TRANSITION #StateOk:
ST08_408_Y54_4.State=STATE_OK

AND gTipImp
END_TRANSITION

TRANSITION #StateOk:
ST08_408_Y54_2.State=STATE_OK

AND gTipImp
END_TRANSITION

TRANSITION #StateOk:
ST08_408_Y54_2.State=STATE_OK

AND gTipImp
END_TRANSITION

TRANSITION CheckCloseDepal:
ST08_405_B53_3.ValveSensor AND	 	(* Rückhaltezylinder links Traystapel Isokörper GST *)
ST08_405_B53_5.ValveSensor AND		(* Rückhaltezylinder rechts Traystapel Isokörper GST *)
gTipImp
END_TRANSITION

TRANSITION #StateOk:
ST08_408_Y54_0.State=STATE_OK

AND gTipImp
END_TRANSITION

TRANSITION with_Motor:
MP.ST08.StapelMotor
END_TRANSITION

TRANSITION Motor_on:
ST08_185_M1.On
END_TRANSITION

TRANSITION busy:
ST08_185_M1.Busy
END_TRANSITION

TRANSITION Done:
ST08_185_M1.Done AND
gTipImp
END_TRANSITION

TRANSITION #StateOk:
ST08_408_Y54_4.State=STATE_OK

AND gTipImp
END_TRANSITION

TRANSITION #StateOk:
ST08_408_Y54_2.State=STATE_OK

AND gTipImp
END_TRANSITION

TRANSITION ExitPosRdy:
ExitPosRdy_T.Q
END_TRANSITION

TRANSITION StateOk:
ST08_406_Y51_2.State=STATE_OK AND
NOT ST00_227_S1.BitInToCheck AND
gTipImp
END_TRANSITION

TRANSITION not_3621:
NOT MP.ST03.SGM_3621
END_TRANSITION

TRANSITION StateOk:
ST08_400_Y52_5.State=STATE_OK AND
ST08_407_Y51_4.State=STATE_OK AND
gTipImp
END_TRANSITION

TRANSITION StateOk:
ST08_408_Y54_4.State =STATE_OK AND
ST08_407_Y51_4.State=STATE_OK AND
gTipImp
END_TRANSITION

TRANSITION Not_Testpart:
NOT TestpartMoveOut
END_TRANSITION

TRANSITION AutoStop:
		ModeSelect.Mode=MODE_AUTO_STOP
OR	ModeSelect.Mode=MODE_STEP_STOP
END_TRANSITION

TRANSITION TrayKompletOut:
NOT ST08_409_B55_5.BitInToCheck AND
gTipImp
END_TRANSITION

TRANSITION InOutlett:
ST08_409_B55_5.BitInToCheck AND
gTipImp
END_TRANSITION

TRANSITION StateOk:
ST08_407_Y51_4.State=STATE_OK AND
NOT ST00_227_S2.BitInToCheck AND
NOT ST00_230_S1.BitInToCheck AND
ST08_408_Y54_0.State=STATE_OK AND
gTipImp
END_TRANSITION

TRANSITION not_3621:
NOT MP.ST03.SGM_3621
END_TRANSITION

TRANSITION StateOk:
(*ST08_408_Y54_4.State=STATE_OK*)

ST08_400_Y52_5.State=STATE_OK AND
gTipImp
END_TRANSITION

TRANSITION StateOk:
ST08_408_Y54_4.State=STATE_OK

AND gTipImp
END_TRANSITION

TRANSITION NOT_gRunEmpty:
NOT gRunEmpty OR
LastTray
END_TRANSITION

TRANSITION WaitTray:
NOT ST08_407_B55_4.BitInToCheck AND	(* Tray in Aufstapelposition eingelaufen STN8 *)
LastTray AND	 (*damit wird im ST08_Process das ausschleusen des halbvollen Blisters bestätigt*)
gTipImp
END_TRANSITION
END_PROGRAM

(* POU Stations/ST_08_Palettierer/ST_08_SFCs/ST08_Process, SFC *)
PROGRAM ST08_Process

VAR_OUTPUT
	SFCCurrentPOU			: STRING:='ST08_Process';
	SFCCurrentStep			: STRING:='';
	FB_CurrentStepHistorie	: FB_CurrentStepHistorie;
	SFCTime					: DINT;
	State   				: StateObject	:= STATE_WAIT;
	Result  				: StateResult;
	ConveyorHQE      	: BOOL;
	ConveyorOut       	: BOOL;
END_VAR
VAR_INPUT
	Start				: BOOL;
END_VAR
VAR
	MsgOK				: BOOL;
	MsgCancel			: BOOL;
	SFCRun				: BOOL;
	SFCTimeStart		: TIME;
	Delay				: TON;
	Delay1				: TON;
	Error				: ErrorStruct;
	(* Userdefinded area *)
	Pal_Ready     		: BOOL;


END_VAR
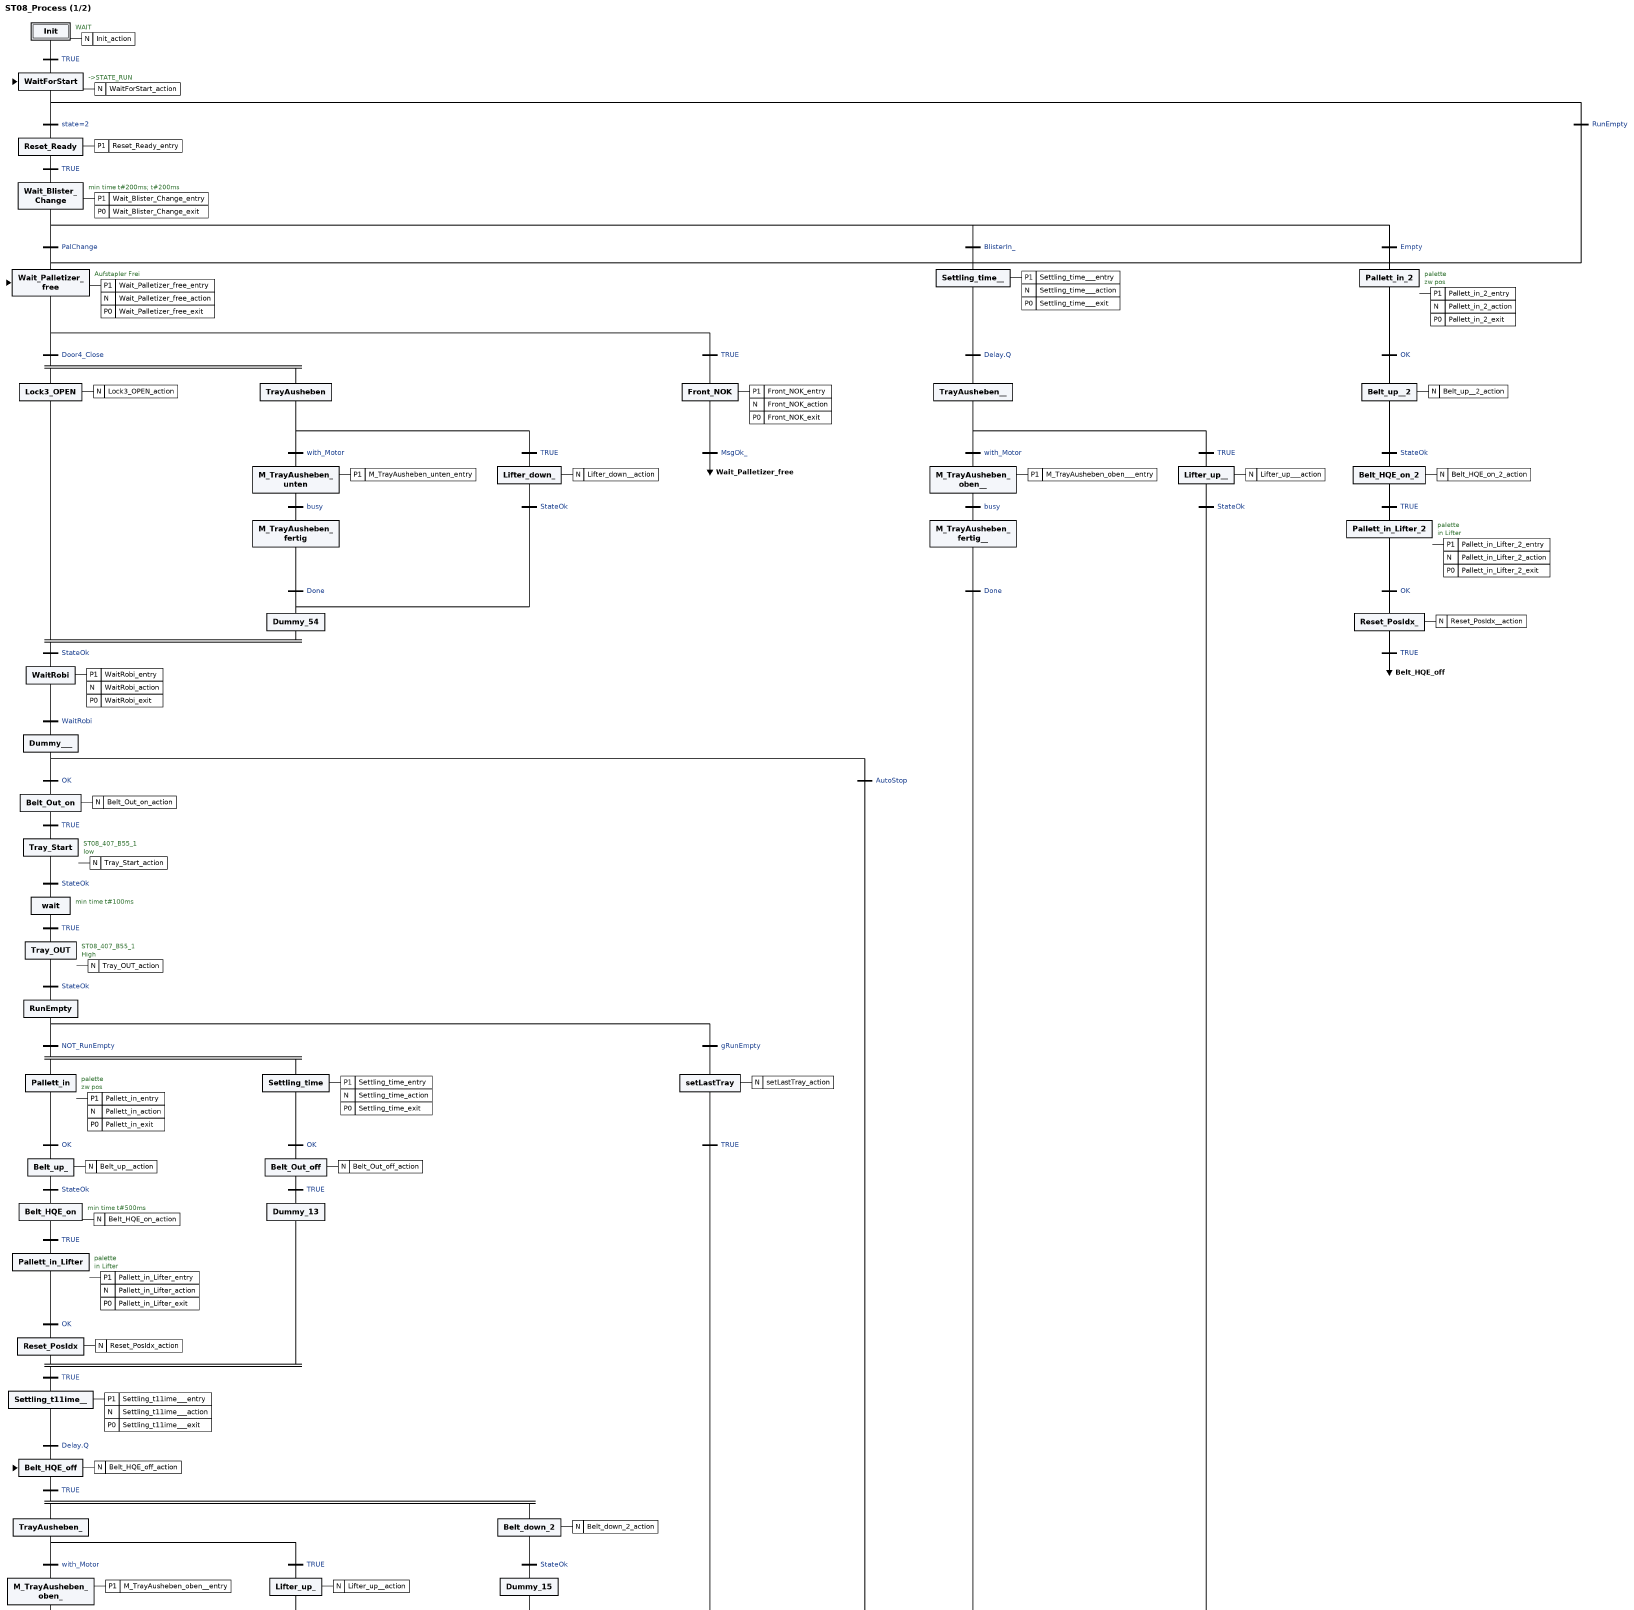
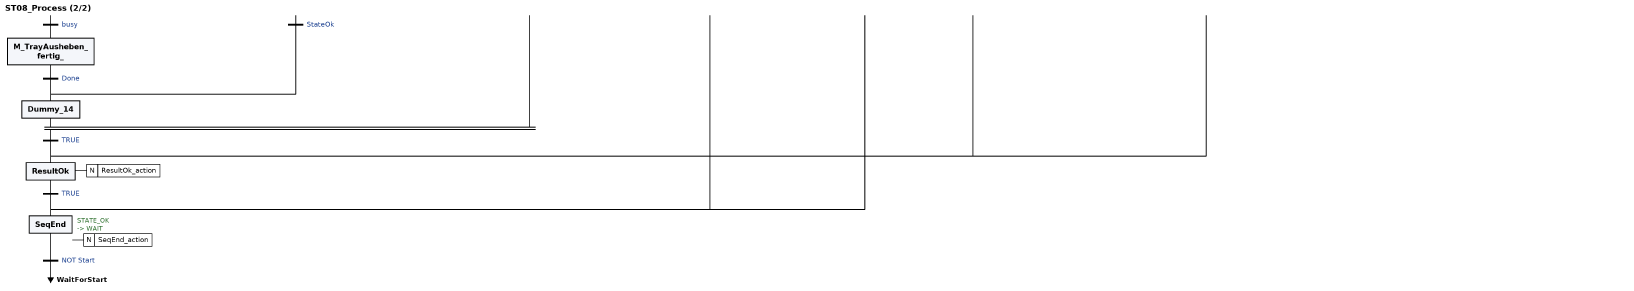
INITIAL_STEP Init: (* WAIT *)
	Init_action(N);
END_STEP
TRANSITION FROM Init TO WaitForStart := TRUE;
END_TRANSITION
STEP WaitForStart: (* ->STATE_RUN *)
	WaitForStart_action(N);
END_STEP
TRANSITION FROM WaitForStart TO Reset_Ready := state=2;
END_TRANSITION
TRANSITION FROM WaitForStart TO Wait_Palletizer_free := RunEmpty;
END_TRANSITION
STEP Reset_Ready:
	Reset_Ready_entry(P1);
END_STEP
TRANSITION FROM Reset_Ready TO Wait_Blister_Change := TRUE;
END_TRANSITION
STEP Wait_Blister_Change: (* min time t#200ms; t#200ms *)
	Wait_Blister_Change_entry(P1);
	Wait_Blister_Change_exit(P0);
END_STEP
TRANSITION FROM Wait_Blister_Change TO Wait_Palletizer_free := PalChange;
END_TRANSITION
TRANSITION FROM Wait_Blister_Change TO Settling_time__ := BlisterIn_;
END_TRANSITION
TRANSITION FROM Wait_Blister_Change TO Pallett_in_2 := Empty;
END_TRANSITION
STEP Wait_Palletizer_free: (* Aufstapler Frei *)
	Wait_Palletizer_free_entry(P1);
	Wait_Palletizer_free_action(N);
	Wait_Palletizer_free_exit(P0);
END_STEP
TRANSITION FROM Wait_Palletizer_free TO (Lock3_OPEN, TrayAusheben) := Door4_Close;
END_TRANSITION
TRANSITION FROM Wait_Palletizer_free TO Front_NOK := TRUE;
END_TRANSITION
STEP Front_NOK:
	Front_NOK_entry(P1);
	Front_NOK_action(N);
	Front_NOK_exit(P0);
END_STEP
TRANSITION FROM Front_NOK TO Wait_Palletizer_free := MsgOk_;
END_TRANSITION
STEP Lock3_OPEN:
	Lock3_OPEN_action(N);
END_STEP
STEP TrayAusheben:
END_STEP
TRANSITION FROM TrayAusheben TO M_TrayAusheben_unten := with_Motor;
END_TRANSITION
TRANSITION FROM TrayAusheben TO Lifter_down_ := TRUE;
END_TRANSITION
STEP M_TrayAusheben_unten:
	M_TrayAusheben_unten_entry(P1);
END_STEP
TRANSITION FROM M_TrayAusheben_unten TO M_TrayAusheben_fertig := busy;
END_TRANSITION
STEP M_TrayAusheben_fertig:
END_STEP
TRANSITION FROM M_TrayAusheben_fertig TO Dummy_54 := Done;
END_TRANSITION
STEP Lifter_down_:
	Lifter_down__action(N);
END_STEP
TRANSITION FROM Lifter_down_ TO Dummy_54 := StateOk;
END_TRANSITION
STEP Dummy_54:
END_STEP
TRANSITION FROM (Lock3_OPEN, Dummy_54) TO WaitRobi := StateOk;
END_TRANSITION
STEP WaitRobi:
	WaitRobi_entry(P1);
	WaitRobi_action(N);
	WaitRobi_exit(P0);
END_STEP
TRANSITION FROM WaitRobi TO Dummy___ := WaitRobi;
END_TRANSITION
STEP Dummy___:
END_STEP
TRANSITION FROM Dummy___ TO Belt_Out_on := OK;
END_TRANSITION
TRANSITION FROM Dummy___ TO SeqEnd := AutoStop;
END_TRANSITION
STEP Belt_Out_on:
	Belt_Out_on_action(N);
END_STEP
TRANSITION FROM Belt_Out_on TO Tray_Start := TRUE;
END_TRANSITION
STEP Tray_Start: (* ST08_407_B55_1 / low *)
	Tray_Start_action(N);
END_STEP
TRANSITION FROM Tray_Start TO wait := StateOk;
END_TRANSITION
STEP wait: (* min time t#100ms *)
END_STEP
TRANSITION FROM wait TO Tray_OUT := TRUE;
END_TRANSITION
STEP Tray_OUT: (* ST08_407_B55_1 / High *)
	Tray_OUT_action(N);
END_STEP
TRANSITION FROM Tray_OUT TO RunEmpty := StateOk;
END_TRANSITION
STEP RunEmpty:
END_STEP
TRANSITION FROM RunEmpty TO (Pallett_in, Settling_time) := NOT_RunEmpty;
END_TRANSITION
TRANSITION FROM RunEmpty TO setLastTray := gRunEmpty;
END_TRANSITION
STEP setLastTray:
	setLastTray_action(N);
END_STEP
TRANSITION FROM setLastTray TO SeqEnd := TRUE;
END_TRANSITION
STEP Pallett_in: (* palette / zw pos *)
	Pallett_in_entry(P1);
	Pallett_in_action(N);
	Pallett_in_exit(P0);
END_STEP
TRANSITION FROM Pallett_in TO Belt_up_ := OK;
END_TRANSITION
STEP Belt_up_:
	Belt_up__action(N);
END_STEP
TRANSITION FROM Belt_up_ TO Belt_HQE_on := StateOk;
END_TRANSITION
STEP Belt_HQE_on: (* min time t#500ms *)
	Belt_HQE_on_action(N);
END_STEP
TRANSITION FROM Belt_HQE_on TO Pallett_in_Lifter := TRUE;
END_TRANSITION
STEP Pallett_in_Lifter: (* palette / in Lifter *)
	Pallett_in_Lifter_entry(P1);
	Pallett_in_Lifter_action(N);
	Pallett_in_Lifter_exit(P0);
END_STEP
TRANSITION FROM Pallett_in_Lifter TO Reset_PosIdx := OK;
END_TRANSITION
STEP Reset_PosIdx:
	Reset_PosIdx_action(N);
END_STEP
STEP Settling_time:
	Settling_time_entry(P1);
	Settling_time_action(N);
	Settling_time_exit(P0);
END_STEP
TRANSITION FROM Settling_time TO Belt_Out_off := OK;
END_TRANSITION
STEP Belt_Out_off:
	Belt_Out_off_action(N);
END_STEP
TRANSITION FROM Belt_Out_off TO Dummy_13 := TRUE;
END_TRANSITION
STEP Dummy_13:
END_STEP
TRANSITION FROM (Reset_PosIdx, Dummy_13) TO Settling_t11ime__ := TRUE;
END_TRANSITION
STEP Settling_t11ime__:
	Settling_t11ime___entry(P1);
	Settling_t11ime___action(N);
	Settling_t11ime___exit(P0);
END_STEP
TRANSITION FROM Settling_t11ime__ TO Belt_HQE_off := Delay.Q;
END_TRANSITION
STEP Belt_HQE_off:
	Belt_HQE_off_action(N);
END_STEP
TRANSITION FROM Belt_HQE_off TO (TrayAusheben_, Belt_down_2) := TRUE;
END_TRANSITION
STEP TrayAusheben_:
END_STEP
TRANSITION FROM TrayAusheben_ TO M_TrayAusheben_oben_ := with_Motor;
END_TRANSITION
TRANSITION FROM TrayAusheben_ TO Lifter_up_ := TRUE;
END_TRANSITION
STEP M_TrayAusheben_oben_:
	M_TrayAusheben_oben__entry(P1);
END_STEP
TRANSITION FROM M_TrayAusheben_oben_ TO M_TrayAusheben_fertig_ := busy;
END_TRANSITION
STEP M_TrayAusheben_fertig_:
END_STEP
TRANSITION FROM M_TrayAusheben_fertig_ TO Dummy_14 := Done;
END_TRANSITION
STEP Lifter_up_:
	Lifter_up__action(N);
END_STEP
TRANSITION FROM Lifter_up_ TO Dummy_14 := StateOk;
END_TRANSITION
STEP Dummy_14:
END_STEP
STEP Belt_down_2:
	Belt_down_2_action(N);
END_STEP
TRANSITION FROM Belt_down_2 TO Dummy_15 := StateOk;
END_TRANSITION
STEP Dummy_15:
END_STEP
TRANSITION FROM (Dummy_14, Dummy_15) TO ResultOk := TRUE;
END_TRANSITION
STEP Settling_time__:
	Settling_time___entry(P1);
	Settling_time___action(N);
	Settling_time___exit(P0);
END_STEP
TRANSITION FROM Settling_time__ TO TrayAusheben__ := Delay.Q;
END_TRANSITION
STEP TrayAusheben__:
END_STEP
TRANSITION FROM TrayAusheben__ TO M_TrayAusheben_oben__ := with_Motor;
END_TRANSITION
TRANSITION FROM TrayAusheben__ TO Lifter_up__ := TRUE;
END_TRANSITION
STEP M_TrayAusheben_oben__:
	M_TrayAusheben_oben___entry(P1);
END_STEP
TRANSITION FROM M_TrayAusheben_oben__ TO M_TrayAusheben_fertig__ := busy;
END_TRANSITION
STEP M_TrayAusheben_fertig__:
END_STEP
TRANSITION FROM M_TrayAusheben_fertig__ TO ResultOk := Done;
END_TRANSITION
STEP Lifter_up__:
	Lifter_up___action(N);
END_STEP
TRANSITION FROM Lifter_up__ TO ResultOk := StateOk;
END_TRANSITION
STEP Pallett_in_2: (* palette / zw pos *)
	Pallett_in_2_entry(P1);
	Pallett_in_2_action(N);
	Pallett_in_2_exit(P0);
END_STEP
TRANSITION FROM Pallett_in_2 TO Belt_up__2 := OK;
END_TRANSITION
STEP Belt_up__2:
	Belt_up__2_action(N);
END_STEP
TRANSITION FROM Belt_up__2 TO Belt_HQE_on_2 := StateOk;
END_TRANSITION
STEP Belt_HQE_on_2:
	Belt_HQE_on_2_action(N);
END_STEP
TRANSITION FROM Belt_HQE_on_2 TO Pallett_in_Lifter_2 := TRUE;
END_TRANSITION
STEP Pallett_in_Lifter_2: (* palette / in Lifter *)
	Pallett_in_Lifter_2_entry(P1);
	Pallett_in_Lifter_2_action(N);
	Pallett_in_Lifter_2_exit(P0);
END_STEP
TRANSITION FROM Pallett_in_Lifter_2 TO Reset_PosIdx_ := OK;
END_TRANSITION
STEP Reset_PosIdx_:
	Reset_PosIdx__action(N);
END_STEP
TRANSITION FROM Reset_PosIdx_ TO Belt_HQE_off := TRUE;
END_TRANSITION
STEP ResultOk:
	ResultOk_action(N);
END_STEP
TRANSITION FROM ResultOk TO SeqEnd := TRUE;
END_TRANSITION
STEP SeqEnd: (* STATE_OK / -> WAIT *)
	SeqEnd_action(N);
END_STEP
TRANSITION FROM SeqEnd TO WaitForStart := NOT Start;
END_TRANSITION

ACTION Init_action:
Start:=FALSE;
State:=STATE_WAIT;
MsgOK:=FALSE;
MsgCancel:=FALSE;
SFCRun:=FALSE;
Pal_Ready:=FALSE;
ConveyorHQE:=FALSE;
ConveyorOut:=FALSE;
END_ACTION

ACTION WaitForStart_action:
IF 	Start OR
	SpecialMode01.State=State_Run OR
	SpecialMode06.State=State_Run THEN
	State:=STATE_RUN;
	Result:=RESULT_NON;
	SFCTimeStart:=TIME();
END_IF
END_ACTION

ACTION Reset_Ready_entry:
(*Pal_Ready:=FALSE;
*);
END_ACTION

ACTION Wait_Blister_Change_entry:
State:=STATE_OK;
END_ACTION

ACTION Wait_Blister_Change_exit:
State:=STATE_RUN;
END_ACTION

ACTION Wait_Palletizer_free_entry:
Pal_Ready:=FALSE;
ProcessMessage01:='';
END_ACTION

ACTION Wait_Palletizer_free_action:
ProcessMessage01:='1IM2';(*St.8 warte auf Palettierer frei und Türe 3 offen*)
END_ACTION

ACTION Wait_Palletizer_free_exit:
ProcessMessage01:='';
END_ACTION

ACTION Front_NOK_entry:
MessageHandler.ClearMessageLines(sVisu:=Visu.Message);
END_ACTION

ACTION Front_NOK_action:
MessageHandler.Msg.ID:='PM202';
MessageHandler.Msg.Name:=ST03_70U3_1.sInit.Description;
MessageHandler.Msg.Text:='Auslauf voll';
MessageHandler.Msg.Color:=Color.blue;
MessageHandler.Msg.Station:=1;


MessageHandler(
	Prio:=2, 							(*1=highest, .. , 4=lowest*)
	Btn1Addr:=ADR(MsgOk),			(*Address of Button1 , if Zero then Button is unvisible*)
	Btn2Addr:=,						(*Address of Button2 , if Zero then Button is unvisible*)
	sVisu:=Visu.Message);
END_ACTION

ACTION Front_NOK_exit:
MsgOk:=FALSE;
MsgCancel:=FALSE;
END_ACTION

ACTION Lock3_OPEN_action:
ST08_406_Y51_2.MoveWork:=TRUE;
END_ACTION

ACTION M_TrayAusheben_unten_entry:
ST08_190_M1.MoveAbs:=TRUE;
ST08_190_M1.Vorgabe_Pos_Abs:=TD.PosTrayAusheben[1].Pos;	(*1=unten, 2=oben, *)
END_ACTION

ACTION Lifter_down__action:
ST08_406_Y52_3.MoveInit:=TRUE;
END_ACTION

ACTION WaitRobi_entry:
Delay(IN:=FALSE);
END_ACTION

ACTION WaitRobi_action:
(*damit beim Leerfahren kein Robi mehr fährt*)
Delay(IN:=
	Robot01.State = STATE_WAIT AND
	Robot01.ActualArea <> 6,
	PT:=t#500ms);
END_ACTION

ACTION WaitRobi_exit:
Delay(IN:=FALSE);
END_ACTION

ACTION Belt_Out_on_action:
ConveyorOut:=TRUE;
END_ACTION

ACTION Tray_Start_action:
ST08_406_B54_6.CheckSignallow:=TRUE;
END_ACTION

ACTION Tray_OUT_action:
ST08_406_B54_6.CheckSignalhigh:=TRUE;
END_ACTION

ACTION setLastTray_action:
ST08_Palletizing.LastTray:=TRUE; (*startet ST08_Palletizing um den letzten halb vollen Tray auszschleusen*)
END_ACTION

ACTION Pallett_in_entry:
ProcessMessage01:='';
END_ACTION

ACTION Pallett_in_action:
ProcessMessage01:='1IM3';(*St.8 warte auf Palette in Zwischen pos HQE*)
END_ACTION

ACTION Pallett_in_exit:
ProcessMessage01:='';
END_ACTION

ACTION Belt_up__action:
ST08_404_Y52_0.MoveWork:=TRUE;
END_ACTION

ACTION Belt_HQE_on_action:
ConveyorHQE:=TRUE;
END_ACTION

ACTION Pallett_in_Lifter_entry:
ProcessMessage01:='';
Delay.IN:=FALSE;
Delay();
END_ACTION

ACTION Pallett_in_Lifter_action:
ProcessMessage01:='1IM4';(*St.8 warte auf Palette in Ausheber*)

Delay.IN:=NOT ST08_406_B54_3.BitInToCheck;
Delay.PT:=T#500ms;
Delay();
END_ACTION

ACTION Pallett_in_Lifter_exit:
ProcessMessage01:='';
END_ACTION

ACTION Reset_PosIdx_action:
PosIdx:=TD.PartsInRoboGripper;
END_ACTION

ACTION Settling_time_entry:
Delay1.IN:=FALSE;
Delay1();
ProcessMessage01:='';
PosIdx:=TD.PartsInRoboGripper;
END_ACTION

ACTION Settling_time_action:
Delay1.IN:=NOT ST08_407_B55_4.BitInToCheck;     (*Blister in Aufstapler*)
Delay1.PT:=T#50ms;
Delay1();

ProcessMessage01:='1IM1';(*St.8 warte auf Palette in Aufstapler*)
END_ACTION

ACTION Settling_time_exit:
ProcessMessage01:='';
END_ACTION

ACTION Belt_Out_off_action:
ConveyorOut:=FALSE;
END_ACTION

ACTION Settling_t11ime___entry:
Delay.IN:=FALSE;
Delay();
ProcessMessage01:='';
END_ACTION

ACTION Settling_t11ime___action:
Delay.IN:=TRUE;     (*Blister in Aufstapler*)
Delay.PT:=T#300ms;
Delay();

ProcessMessage01:='1IM1';(*St.8 warte auf Palette in Aufstapler*)
END_ACTION

ACTION Settling_t11ime___exit:
ProcessMessage01:='';
END_ACTION

ACTION Belt_HQE_off_action:
ConveyorHQE:=FALSE;
END_ACTION

ACTION M_TrayAusheben_oben__entry:
ST08_190_M1.MoveAbs:=TRUE;
ST08_190_M1.Vorgabe_Pos_Abs:=TD.PosTrayAusheben[2].Pos;	(*1=unten, 2=oben, *)
END_ACTION

ACTION Lifter_up__action:
ST08_406_Y52_3.MoveWork:=TRUE;
END_ACTION

ACTION Belt_down_2_action:
ST08_404_Y52_0.MoveInit:=TRUE;
END_ACTION

ACTION Settling_time___entry:
Delay.IN:=FALSE;
Delay();
ProcessMessage01:='';
END_ACTION

ACTION Settling_time___action:
Delay.IN:=TRUE;     (*Blister in Aufstapler*)
Delay.PT:=T#1s;
Delay();

ProcessMessage01:='1IM1';(*St.8 warte auf Palette in Aufstapler*)
END_ACTION

ACTION Settling_time___exit:
ProcessMessage01:='';
END_ACTION

ACTION M_TrayAusheben_oben___entry:
ST08_190_M1.MoveAbs:=TRUE;
ST08_190_M1.Vorgabe_Pos_Abs:=TD.PosTrayAusheben[2].Pos;	(*1=unten, 2=oben, *)
END_ACTION

ACTION Lifter_up___action:
ST08_406_Y52_3.MoveWork:=TRUE;
END_ACTION

ACTION Pallett_in_2_entry:
ProcessMessage01:='';
END_ACTION

ACTION Pallett_in_2_action:
ProcessMessage01:='1IM3';(*St.8 warte auf Palette in Zwischen pos HQE*)
END_ACTION

ACTION Pallett_in_2_exit:
Pal_Ready:=FALSE;
ProcessMessage01:='';
END_ACTION

ACTION Belt_up__2_action:
ST08_404_Y52_0.MoveWork:=TRUE;
END_ACTION

ACTION Belt_HQE_on_2_action:
ConveyorHQE:=TRUE;
END_ACTION

ACTION Pallett_in_Lifter_2_entry:
ProcessMessage01:='';
Delay.IN:=FALSE;
Delay();
END_ACTION

ACTION Pallett_in_Lifter_2_action:
ProcessMessage01:='1IM4';(*St.8 warte auf Palette in Ausheber*)

Delay.IN:=NOT ST08_406_B54_3.BitInToCheck;
Delay.PT:=T#150ms;
Delay();
END_ACTION

ACTION Pallett_in_Lifter_2_exit:
ProcessMessage01:='';
END_ACTION

ACTION Reset_PosIdx__action:
PosIdx:=TD.PartsInRoboGripper;
END_ACTION

ACTION ResultOk_action:
Result:=RESULT_OK;
END_ACTION

ACTION SeqEnd_action:
IF 	State=STATE_RUN THEN
	SFCTime:=TIME_TO_DINT(TIME()-SFCTimeStart);
	State:=STATE_OK;
END_IF

IF 	NOT Start THEN
	State:=STATE_WAIT;
	Pal_Ready:=TRUE;
END_IF
END_ACTION

TRANSITION RunEmpty:
gRunEmpty AND
ST08_Palletizing.WaitLastTray AND
NOT ST08_Palletizing.LastTray
END_TRANSITION

TRANSITION PalChange:
TD.PartsInBlisterInlet < PosIdx  OR
(ST08_Palletizing.TestpartMoveOut AND
ST08_Palletizing.State = State_Wait) OR
(NOT MP.ST08.TrayAushebenMotor AND SpecialMode01.State=State_Run AND ST08_406_Y52_3.WorkPosition ) OR
(MP.ST08.TrayAushebenMotor AND SpecialMode01.State=State_Run AND ABS(ST08_190_M1.sPos.ist - TD.PosTrayAusheben[2].Pos) < 0.5) (*1=unten, 2=oben, *)
END_TRANSITION

TRANSITION Door4_Close:
(MP.ST03.SGM_3621 OR
ST08_407_B55_3.ValveSensor)	(* Hubtüre 4 Auslauf STN8 AST (ValveSensor) *)
AND  ST08_409_B55_5.BitInToCheck (* kein Stau im Auslauf *)
END_TRANSITION

TRANSITION MsgOk_:
((MP.ST03.SGM_3621 OR
ST08_407_B55_3.ValveSensor)	AND (* Hubtüre 4 Auslauf STN8 AST (ValveSensor) *)
ST08_409_B55_5.BitInToCheck) (* kein Stau im Auslauf *)

OR MsgOk
END_TRANSITION

TRANSITION with_Motor:
MP.ST08.TrayAushebenMotor
END_TRANSITION

TRANSITION busy:
ST08_190_M1.Busy
END_TRANSITION

TRANSITION Done:
ST08_190_M1.Done
END_TRANSITION

TRANSITION StateOk:
ST08_406_Y52_3.State=STATE_OK
END_TRANSITION

TRANSITION StateOk:
ST08_406_Y51_2.State=STATE_OK AND
(ST08_406_Y52_3.State=STATE_OK OR
ST08_190_M1.Done)
END_TRANSITION

TRANSITION WaitRobi:
Delay.Q OR
NOT gRunEmpty
END_TRANSITION

TRANSITION OK:
ST08_407_B55_4.BitInToCheck   (*kein Tray in Aufstapler*)
AND ST08_406_Y51_2.WorkPosition (*Tür 3 offen*)
AND ST08_406_B54_6.BitInToCheck (*kein Tray auf Bandstrecke*)
AND NOT ST08_Palletizing.LockInlett
END_TRANSITION

TRANSITION AutoStop:
		ModeSelect.Mode=MODE_AUTO_STOP
OR	ModeSelect.Mode=MODE_STEP_STOP
END_TRANSITION

TRANSITION StateOk:
ST08_406_B54_6.State=STATE_OK
END_TRANSITION

TRANSITION StateOk:
ST08_406_B54_6.State=STATE_OK
END_TRANSITION

TRANSITION NOT_RunEmpty:
NOT gRunEmpty AND
gTipImp
END_TRANSITION

TRANSITION OK:
NOT ST08_406_B54_0.BitInToCheck
END_TRANSITION

TRANSITION StateOk:
ST08_404_Y52_0.State=STATE_OK
END_TRANSITION

TRANSITION OK:
Delay.Q
END_TRANSITION

TRANSITION OK:
Delay1.Q
END_TRANSITION

TRANSITION with_Motor:
MP.ST08.TrayAushebenMotor
END_TRANSITION

TRANSITION busy:
ST08_190_M1.Busy
END_TRANSITION

TRANSITION Done:
ST08_190_M1.Done
END_TRANSITION

TRANSITION StateOk:
ST08_406_Y52_3.State=STATE_OK
END_TRANSITION

TRANSITION StateOk:
ST08_404_Y52_0.State=STATE_OK
END_TRANSITION

TRANSITION BlisterIn_:
(ST08_406_B54_3.BitInToCheck=FALSE OR		(*Ausheber Trays in Entnahmepos. STN8*)
(NOT MP.ST08.TrayAushebenMotor AND ST08_406_Y52_3.WorkPosition) OR
(MP.ST08.TrayAushebenMotor AND ABS(ST08_190_M1.sPos.ist - TD.PosTrayAusheben[2].Pos) < 0.5)) AND (*1=unten, 2=oben, *)
NOT ST08_Palletizing.TestpartMoveOut
END_TRANSITION

TRANSITION with_Motor:
MP.ST08.TrayAushebenMotor
END_TRANSITION

TRANSITION busy:
ST08_190_M1.Busy
END_TRANSITION

TRANSITION Done:
ST08_190_M1.Done
END_TRANSITION

TRANSITION StateOk:
ST08_406_Y52_3.State=STATE_OK
END_TRANSITION

TRANSITION Empty:
ST08_406_B54_3.BitInToCheck AND
NOT ST08_406_B54_0.BitInToCheck AND
((NOT MP.ST08.TrayAushebenMotor AND ST08_406_Y52_3.InitPosition) OR
(MP.ST08.TrayAushebenMotor AND ABS(ST08_190_M1.sPos.ist - TD.PosTrayAusheben[1].Pos) < 0.5)) (*1=unten, 2=oben, *)
END_TRANSITION

TRANSITION OK:
ST08_406_B54_0.BitInToCheck=FALSE
END_TRANSITION

TRANSITION StateOk:
ST08_404_Y52_0.State=STATE_OK
END_TRANSITION

TRANSITION OK:
Delay.Q
END_TRANSITION
END_PROGRAM

(* POU Stations/ST_02_RT_Tampondrucker/ST02_SFCs/ST02_Main, SFC *)
 PROGRAM ST02_Main
VAR_OUTPUT
	SFCCurrentPOU		: STRING:='ST02_Main';
	SFCCurrentStep		: STRING:='';
	FB_CurrentStepHistorie: FB_CurrentStepHistorie;
	SFCTime				: DINT;
	State   			: StateObject	:= STATE_WAIT;
	Result  			: StateResult;

END_VAR
VAR_INPUT
	Start				: BOOL;
END_VAR
VAR
	MsgOK				: BOOL;
	MsgCancel			: BOOL;
	SFCRun				: BOOL;
	SFCTimeStart		: TIME;
	(* Userdefinded area *)
	i					: INT;
	RepeatCounter		: INT;
	NokCounter			: INT;
	NokCounterPercent	: INT;
  	NokPercent   		: ARRAY[1..100] OF BOOL;
	turn_done			: BOOL;
	ResultBuffer		: ARRAY[1..10] OF DINT;
	LoopCounter			: DINT;	(* Anzahl Dummy *)

END_VAR
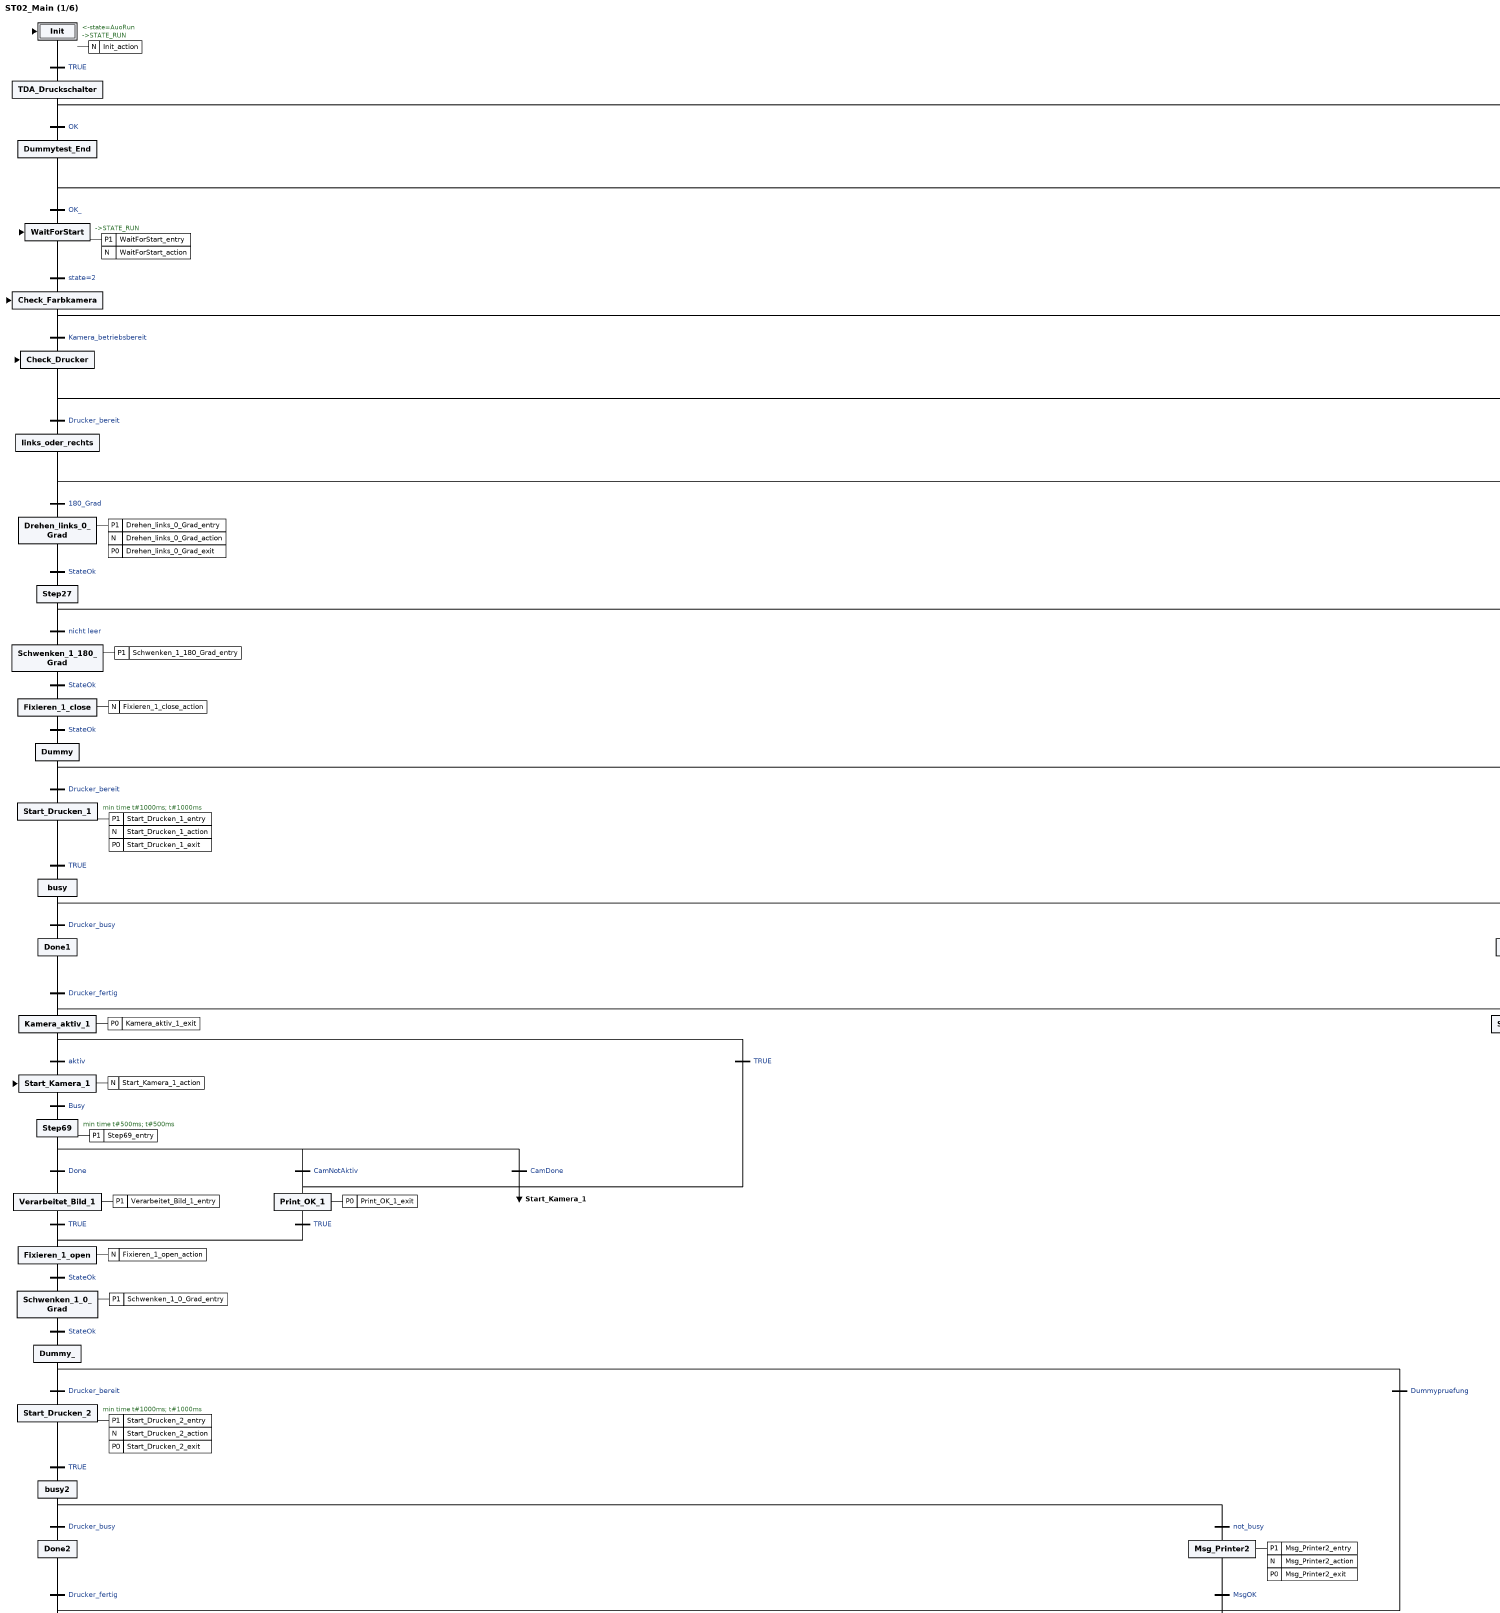
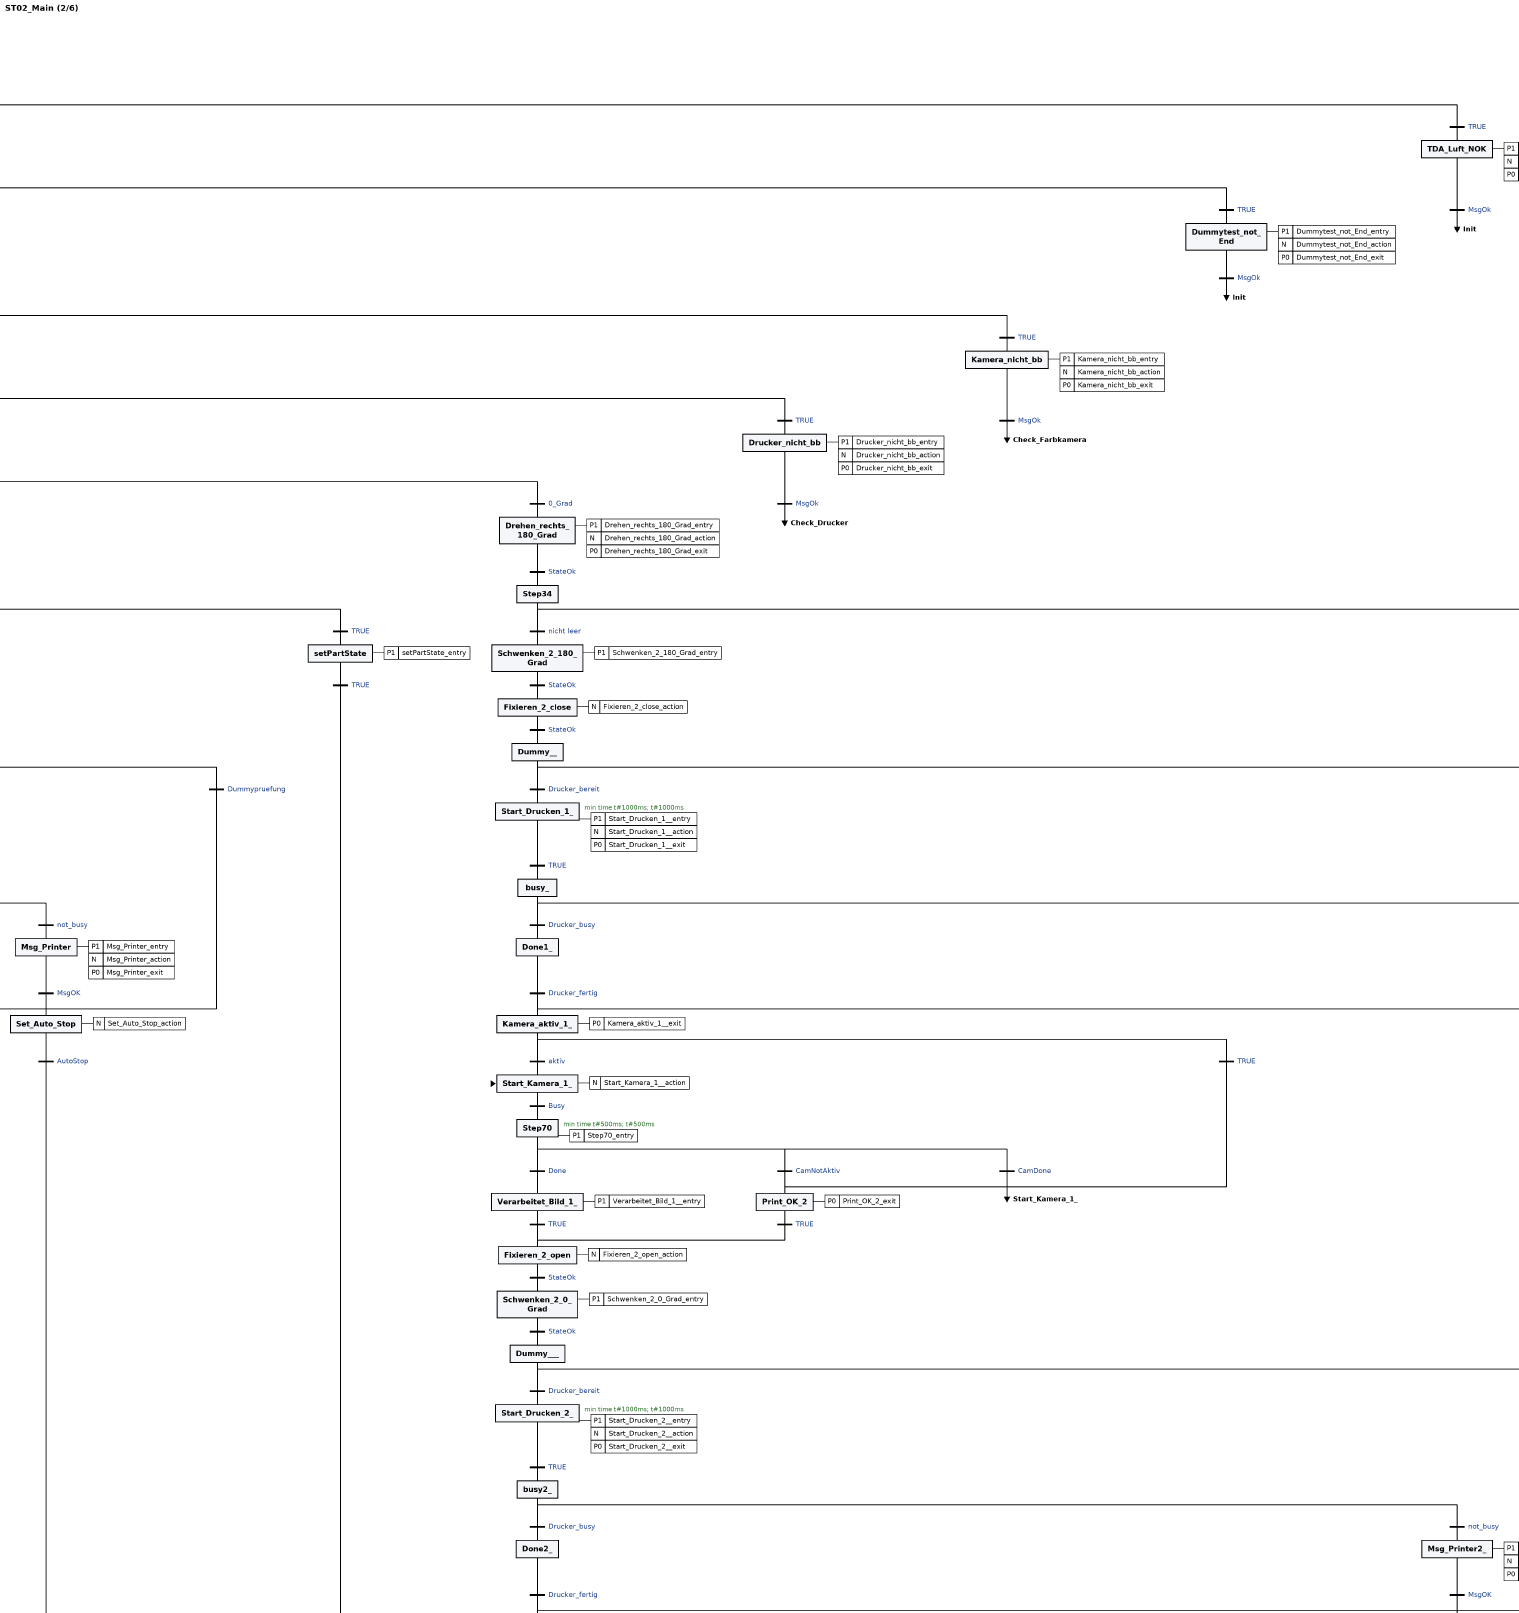
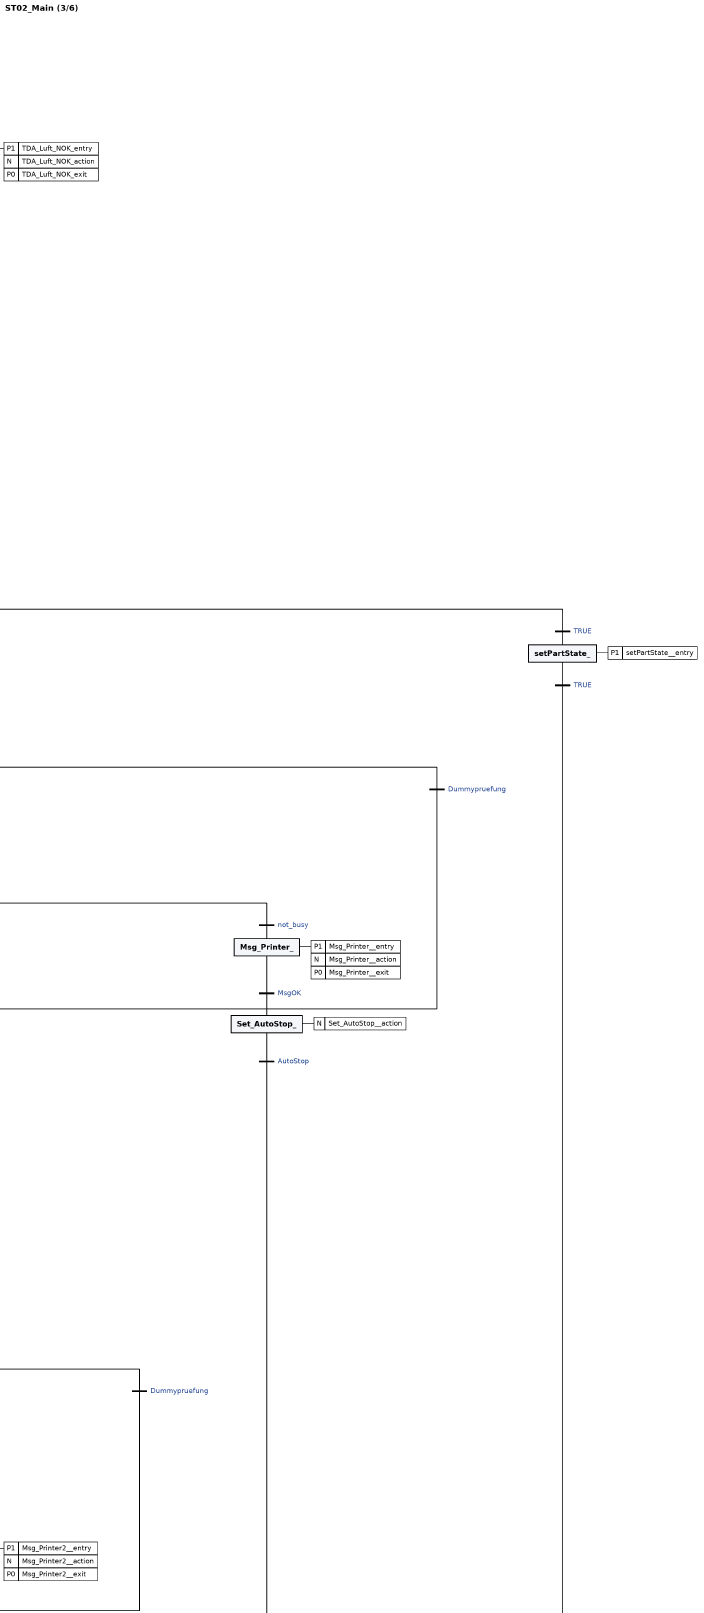
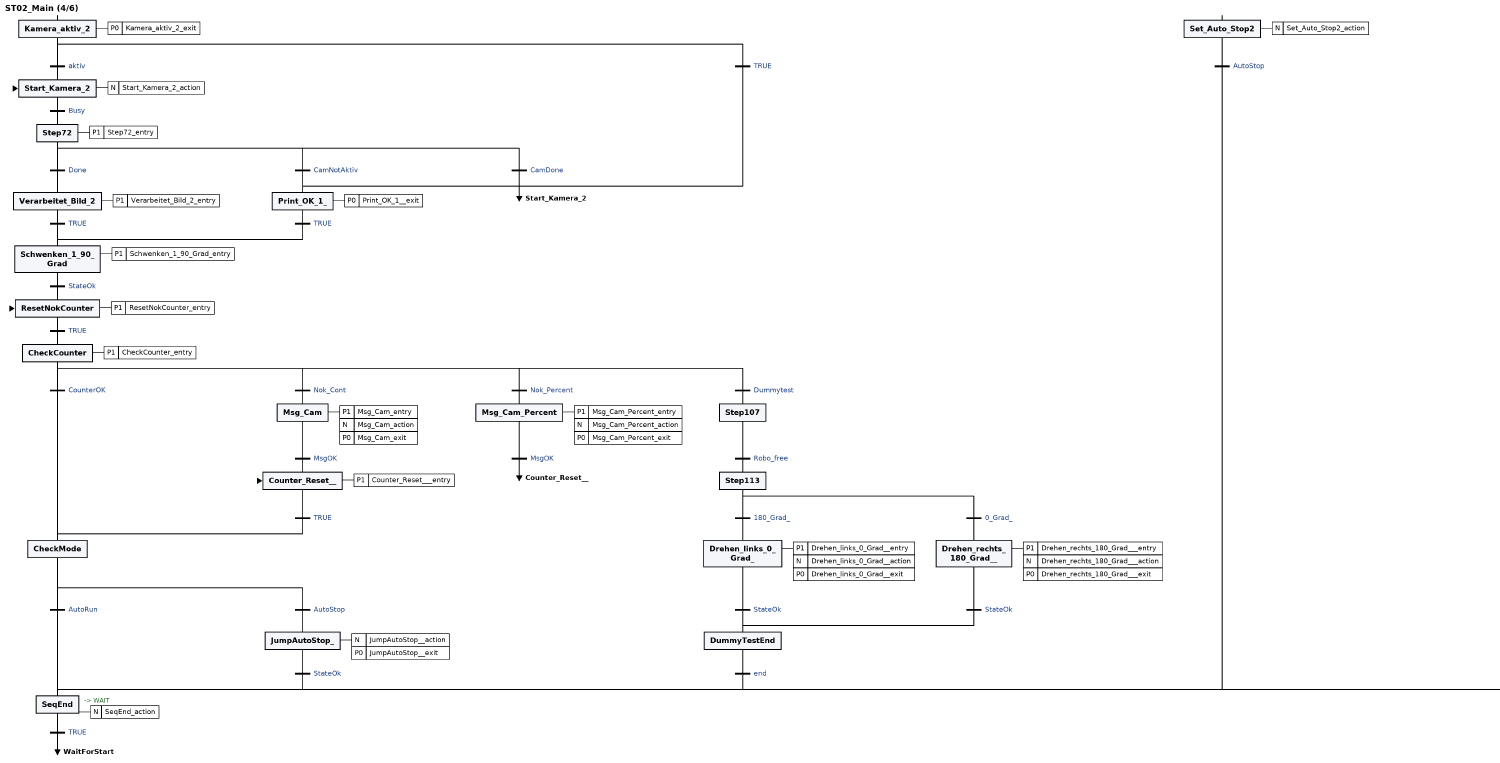
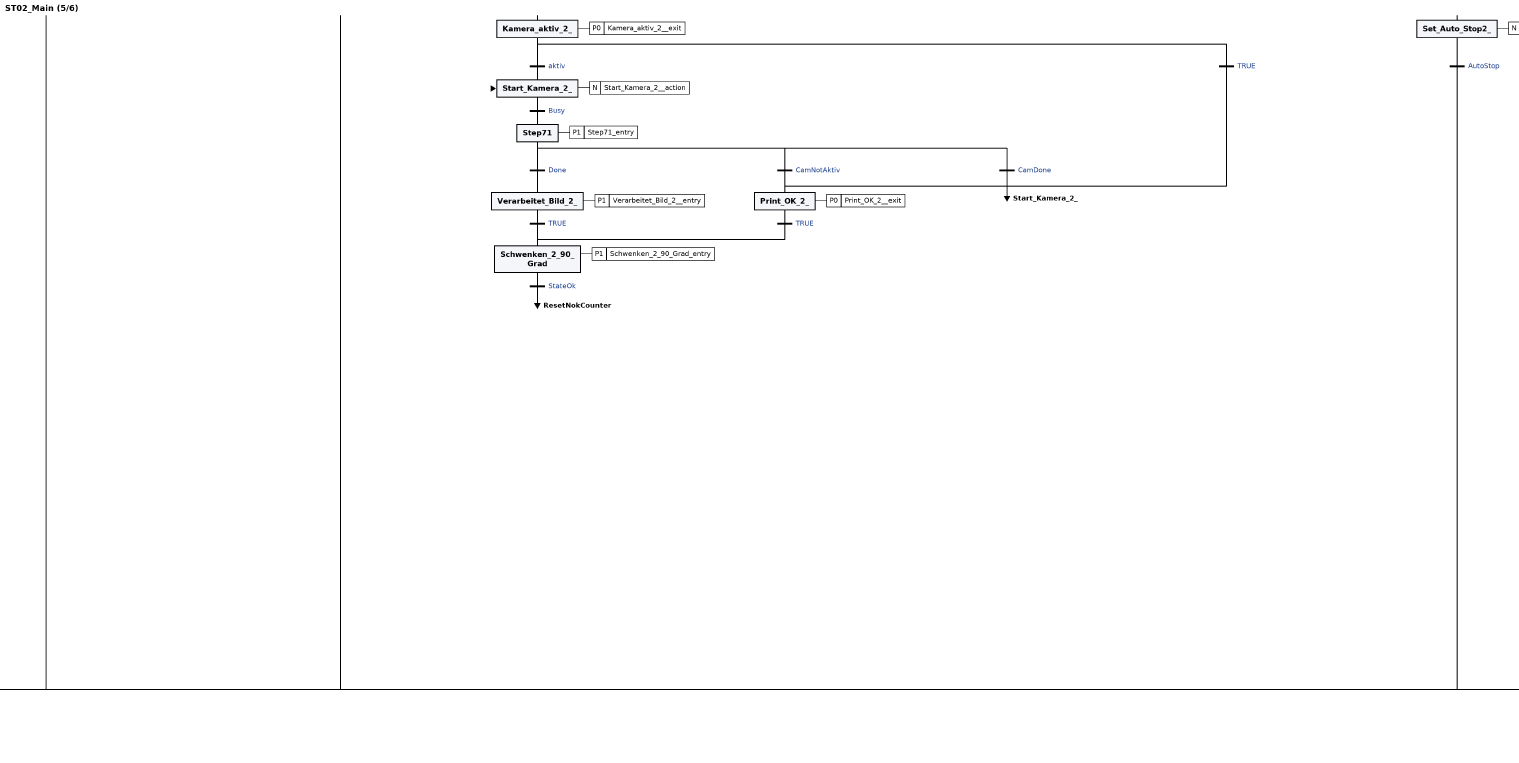
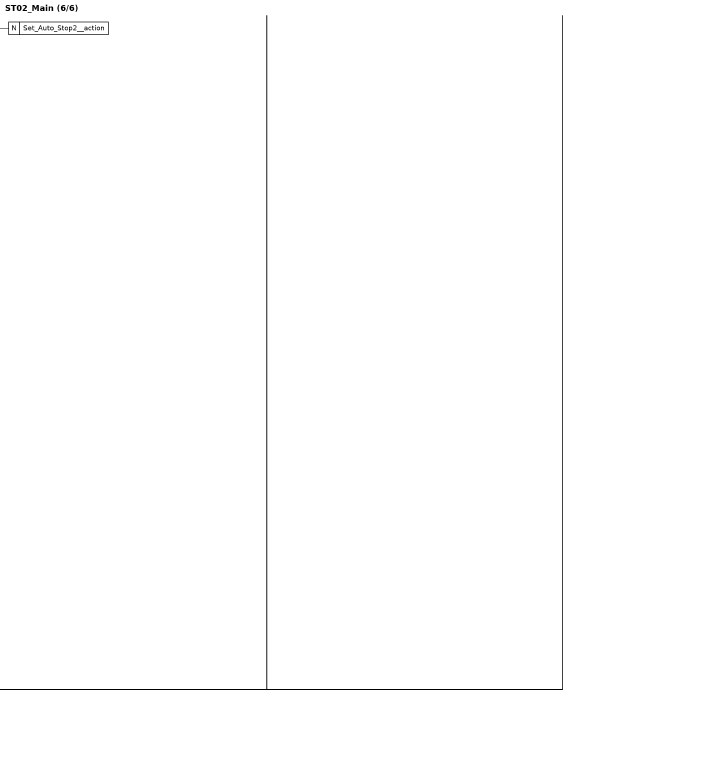
INITIAL_STEP Init: (* <-state=AuoRun / ->STATE_RUN *)
	Init_action(N);
END_STEP
TRANSITION FROM Init TO TDA_Druckschalter := TRUE;
END_TRANSITION
STEP TDA_Druckschalter:
END_STEP
TRANSITION FROM TDA_Druckschalter TO Dummytest_End := OK;
END_TRANSITION
TRANSITION FROM TDA_Druckschalter TO TDA_Luft_NOK := TRUE;
END_TRANSITION
STEP Dummytest_End:
END_STEP
TRANSITION FROM Dummytest_End TO WaitForStart := OK_;
END_TRANSITION
TRANSITION FROM Dummytest_End TO Dummytest_not_End := TRUE;
END_TRANSITION
STEP Dummytest_not_End:
	Dummytest_not_End_entry(P1);
	Dummytest_not_End_action(N);
	Dummytest_not_End_exit(P0);
END_STEP
TRANSITION FROM Dummytest_not_End TO Init := MsgOk;
END_TRANSITION
STEP TDA_Luft_NOK:
	TDA_Luft_NOK_entry(P1);
	TDA_Luft_NOK_action(N);
	TDA_Luft_NOK_exit(P0);
END_STEP
TRANSITION FROM TDA_Luft_NOK TO Init := MsgOk;
END_TRANSITION
STEP WaitForStart: (* ->STATE_RUN *)
	WaitForStart_entry(P1);
	WaitForStart_action(N);
END_STEP
TRANSITION FROM WaitForStart TO Check_Farbkamera := state=2;
END_TRANSITION
STEP Check_Farbkamera:
END_STEP
TRANSITION FROM Check_Farbkamera TO Check_Drucker := Kamera_betriebsbereit;
END_TRANSITION
TRANSITION FROM Check_Farbkamera TO Kamera_nicht_bb := TRUE;
END_TRANSITION
STEP Kamera_nicht_bb:
	Kamera_nicht_bb_entry(P1);
	Kamera_nicht_bb_action(N);
	Kamera_nicht_bb_exit(P0);
END_STEP
TRANSITION FROM Kamera_nicht_bb TO Check_Farbkamera := MsgOk;
END_TRANSITION
STEP Check_Drucker:
END_STEP
TRANSITION FROM Check_Drucker TO links_oder_rechts := Drucker_bereit;
END_TRANSITION
TRANSITION FROM Check_Drucker TO Drucker_nicht_bb := TRUE;
END_TRANSITION
STEP Drucker_nicht_bb:
	Drucker_nicht_bb_entry(P1);
	Drucker_nicht_bb_action(N);
	Drucker_nicht_bb_exit(P0);
END_STEP
TRANSITION FROM Drucker_nicht_bb TO Check_Drucker := MsgOk;
END_TRANSITION
STEP links_oder_rechts:
END_STEP
TRANSITION FROM links_oder_rechts TO Drehen_links_0_Grad := 180_Grad;
END_TRANSITION
TRANSITION FROM links_oder_rechts TO Drehen_rechts_180_Grad := 0_Grad;
END_TRANSITION
STEP Drehen_links_0_Grad:
	Drehen_links_0_Grad_entry(P1);
	Drehen_links_0_Grad_action(N);
	Drehen_links_0_Grad_exit(P0);
END_STEP
TRANSITION FROM Drehen_links_0_Grad TO Step27 := StateOk;
END_TRANSITION
STEP Step27:
END_STEP
TRANSITION FROM Step27 TO Schwenken_1_180_Grad := nicht leer;
END_TRANSITION
TRANSITION FROM Step27 TO setPartState := TRUE;
END_TRANSITION
STEP setPartState:
	setPartState_entry(P1);
END_STEP
TRANSITION FROM setPartState TO SeqEnd := TRUE;
END_TRANSITION
STEP Schwenken_1_180_Grad:
	Schwenken_1_180_Grad_entry(P1);
END_STEP
TRANSITION FROM Schwenken_1_180_Grad TO Fixieren_1_close := StateOk;
END_TRANSITION
STEP Fixieren_1_close:
	Fixieren_1_close_action(N);
END_STEP
TRANSITION FROM Fixieren_1_close TO Dummy := StateOk;
END_TRANSITION
STEP Dummy:
END_STEP
TRANSITION FROM Dummy TO Start_Drucken_1 := Drucker_bereit;
END_TRANSITION
TRANSITION FROM Dummy TO Kamera_aktiv_1 := Dummypruefung;
END_TRANSITION
STEP Start_Drucken_1: (* min time t#1000ms; t#1000ms *)
	Start_Drucken_1_entry(P1);
	Start_Drucken_1_action(N);
	Start_Drucken_1_exit(P0);
END_STEP
TRANSITION FROM Start_Drucken_1 TO busy := TRUE;
END_TRANSITION
STEP busy:
END_STEP
TRANSITION FROM busy TO Done1 := Drucker_busy;
END_TRANSITION
TRANSITION FROM busy TO Msg_Printer := not_busy;
END_TRANSITION
STEP Msg_Printer:
	Msg_Printer_entry(P1);
	Msg_Printer_action(N);
	Msg_Printer_exit(P0);
END_STEP
TRANSITION FROM Msg_Printer TO Set_Auto_Stop := MsgOK;
END_TRANSITION
STEP Set_Auto_Stop:
	Set_Auto_Stop_action(N);
END_STEP
TRANSITION FROM Set_Auto_Stop TO SeqEnd := AutoStop;
END_TRANSITION
STEP Done1:
END_STEP
TRANSITION FROM Done1 TO Kamera_aktiv_1 := Drucker_fertig;
END_TRANSITION
STEP Kamera_aktiv_1:
	Kamera_aktiv_1_exit(P0);
END_STEP
TRANSITION FROM Kamera_aktiv_1 TO Start_Kamera_1 := aktiv;
END_TRANSITION
TRANSITION FROM Kamera_aktiv_1 TO Print_OK_1 := TRUE;
END_TRANSITION
STEP Start_Kamera_1:
	Start_Kamera_1_action(N);
END_STEP
TRANSITION FROM Start_Kamera_1 TO Step69 := Busy;
END_TRANSITION
STEP Step69: (* min time t#500ms; t#500ms *)
	Step69_entry(P1);
END_STEP
TRANSITION FROM Step69 TO Verarbeitet_Bild_1 := Done;
END_TRANSITION
TRANSITION FROM Step69 TO Print_OK_1 := CamNotAktiv;
END_TRANSITION
TRANSITION FROM Step69 TO Start_Kamera_1 := CamDone;
END_TRANSITION
STEP Verarbeitet_Bild_1:
	Verarbeitet_Bild_1_entry(P1);
END_STEP
TRANSITION FROM Verarbeitet_Bild_1 TO Fixieren_1_open := TRUE;
END_TRANSITION
STEP Print_OK_1:
	Print_OK_1_exit(P0);
END_STEP
TRANSITION FROM Print_OK_1 TO Fixieren_1_open := TRUE;
END_TRANSITION
STEP Fixieren_1_open:
	Fixieren_1_open_action(N);
END_STEP
TRANSITION FROM Fixieren_1_open TO Schwenken_1_0_Grad := StateOk;
END_TRANSITION
STEP Schwenken_1_0_Grad:
	Schwenken_1_0_Grad_entry(P1);
END_STEP
TRANSITION FROM Schwenken_1_0_Grad TO Dummy_ := StateOk;
END_TRANSITION
STEP Dummy_:
END_STEP
TRANSITION FROM Dummy_ TO Start_Drucken_2 := Drucker_bereit;
END_TRANSITION
TRANSITION FROM Dummy_ TO Kamera_aktiv_2 := Dummypruefung;
END_TRANSITION
STEP Start_Drucken_2: (* min time t#1000ms; t#1000ms *)
	Start_Drucken_2_entry(P1);
	Start_Drucken_2_action(N);
	Start_Drucken_2_exit(P0);
END_STEP
TRANSITION FROM Start_Drucken_2 TO busy2 := TRUE;
END_TRANSITION
STEP busy2:
END_STEP
TRANSITION FROM busy2 TO Done2 := Drucker_busy;
END_TRANSITION
TRANSITION FROM busy2 TO Msg_Printer2 := not_busy;
END_TRANSITION
STEP Msg_Printer2:
	Msg_Printer2_entry(P1);
	Msg_Printer2_action(N);
	Msg_Printer2_exit(P0);
END_STEP
TRANSITION FROM Msg_Printer2 TO Set_Auto_Stop2 := MsgOK;
END_TRANSITION
STEP Set_Auto_Stop2:
	Set_Auto_Stop2_action(N);
END_STEP
TRANSITION FROM Set_Auto_Stop2 TO SeqEnd := AutoStop;
END_TRANSITION
STEP Done2:
END_STEP
TRANSITION FROM Done2 TO Kamera_aktiv_2 := Drucker_fertig;
END_TRANSITION
STEP Kamera_aktiv_2:
	Kamera_aktiv_2_exit(P0);
END_STEP
TRANSITION FROM Kamera_aktiv_2 TO Start_Kamera_2 := aktiv;
END_TRANSITION
TRANSITION FROM Kamera_aktiv_2 TO Print_OK_1_ := TRUE;
END_TRANSITION
STEP Start_Kamera_2:
	Start_Kamera_2_action(N);
END_STEP
TRANSITION FROM Start_Kamera_2 TO Step72 := Busy;
END_TRANSITION
STEP Step72:
	Step72_entry(P1);
END_STEP
TRANSITION FROM Step72 TO Verarbeitet_Bild_2 := Done;
END_TRANSITION
TRANSITION FROM Step72 TO Print_OK_1_ := CamNotAktiv;
END_TRANSITION
TRANSITION FROM Step72 TO Start_Kamera_2 := CamDone;
END_TRANSITION
STEP Verarbeitet_Bild_2:
	Verarbeitet_Bild_2_entry(P1);
END_STEP
TRANSITION FROM Verarbeitet_Bild_2 TO Schwenken_1_90_Grad := TRUE;
END_TRANSITION
STEP Print_OK_1_:
	Print_OK_1__exit(P0);
END_STEP
TRANSITION FROM Print_OK_1_ TO Schwenken_1_90_Grad := TRUE;
END_TRANSITION
STEP Schwenken_1_90_Grad:
	Schwenken_1_90_Grad_entry(P1);
END_STEP
TRANSITION FROM Schwenken_1_90_Grad TO ResetNokCounter := StateOk;
END_TRANSITION
STEP ResetNokCounter:
	ResetNokCounter_entry(P1);
END_STEP
TRANSITION FROM ResetNokCounter TO CheckCounter := TRUE;
END_TRANSITION
STEP Drehen_rechts_180_Grad:
	Drehen_rechts_180_Grad_entry(P1);
	Drehen_rechts_180_Grad_action(N);
	Drehen_rechts_180_Grad_exit(P0);
END_STEP
TRANSITION FROM Drehen_rechts_180_Grad TO Step34 := StateOk;
END_TRANSITION
STEP Step34:
END_STEP
TRANSITION FROM Step34 TO Schwenken_2_180_Grad := nicht leer;
END_TRANSITION
TRANSITION FROM Step34 TO setPartState_ := TRUE;
END_TRANSITION
STEP setPartState_:
	setPartState__entry(P1);
END_STEP
TRANSITION FROM setPartState_ TO SeqEnd := TRUE;
END_TRANSITION
STEP Schwenken_2_180_Grad:
	Schwenken_2_180_Grad_entry(P1);
END_STEP
TRANSITION FROM Schwenken_2_180_Grad TO Fixieren_2_close := StateOk;
END_TRANSITION
STEP Fixieren_2_close:
	Fixieren_2_close_action(N);
END_STEP
TRANSITION FROM Fixieren_2_close TO Dummy__ := StateOk;
END_TRANSITION
STEP Dummy__:
END_STEP
TRANSITION FROM Dummy__ TO Start_Drucken_1_ := Drucker_bereit;
END_TRANSITION
TRANSITION FROM Dummy__ TO Kamera_aktiv_1_ := Dummypruefung;
END_TRANSITION
STEP Start_Drucken_1_: (* min time t#1000ms; t#1000ms *)
	Start_Drucken_1__entry(P1);
	Start_Drucken_1__action(N);
	Start_Drucken_1__exit(P0);
END_STEP
TRANSITION FROM Start_Drucken_1_ TO busy_ := TRUE;
END_TRANSITION
STEP busy_:
END_STEP
TRANSITION FROM busy_ TO Done1_ := Drucker_busy;
END_TRANSITION
TRANSITION FROM busy_ TO Msg_Printer_ := not_busy;
END_TRANSITION
STEP Msg_Printer_:
	Msg_Printer__entry(P1);
	Msg_Printer__action(N);
	Msg_Printer__exit(P0);
END_STEP
TRANSITION FROM Msg_Printer_ TO Set_AutoStop_ := MsgOK;
END_TRANSITION
STEP Set_AutoStop_:
	Set_AutoStop__action(N);
END_STEP
TRANSITION FROM Set_AutoStop_ TO SeqEnd := AutoStop;
END_TRANSITION
STEP Done1_:
END_STEP
TRANSITION FROM Done1_ TO Kamera_aktiv_1_ := Drucker_fertig;
END_TRANSITION
STEP Kamera_aktiv_1_:
	Kamera_aktiv_1__exit(P0);
END_STEP
TRANSITION FROM Kamera_aktiv_1_ TO Start_Kamera_1_ := aktiv;
END_TRANSITION
TRANSITION FROM Kamera_aktiv_1_ TO Print_OK_2 := TRUE;
END_TRANSITION
STEP Start_Kamera_1_:
	Start_Kamera_1__action(N);
END_STEP
TRANSITION FROM Start_Kamera_1_ TO Step70 := Busy;
END_TRANSITION
STEP Step70: (* min time t#500ms; t#500ms *)
	Step70_entry(P1);
END_STEP
TRANSITION FROM Step70 TO Verarbeitet_Bild_1_ := Done;
END_TRANSITION
TRANSITION FROM Step70 TO Print_OK_2 := CamNotAktiv;
END_TRANSITION
TRANSITION FROM Step70 TO Start_Kamera_1_ := CamDone;
END_TRANSITION
STEP Verarbeitet_Bild_1_:
	Verarbeitet_Bild_1__entry(P1);
END_STEP
TRANSITION FROM Verarbeitet_Bild_1_ TO Fixieren_2_open := TRUE;
END_TRANSITION
STEP Print_OK_2:
	Print_OK_2_exit(P0);
END_STEP
TRANSITION FROM Print_OK_2 TO Fixieren_2_open := TRUE;
END_TRANSITION
STEP Fixieren_2_open:
	Fixieren_2_open_action(N);
END_STEP
TRANSITION FROM Fixieren_2_open TO Schwenken_2_0_Grad := StateOk;
END_TRANSITION
STEP Schwenken_2_0_Grad:
	Schwenken_2_0_Grad_entry(P1);
END_STEP
TRANSITION FROM Schwenken_2_0_Grad TO Dummy___ := StateOk;
END_TRANSITION
STEP Dummy___:
END_STEP
TRANSITION FROM Dummy___ TO Start_Drucken_2_ := Drucker_bereit;
END_TRANSITION
TRANSITION FROM Dummy___ TO Kamera_aktiv_2_ := Dummypruefung;
END_TRANSITION
STEP Start_Drucken_2_: (* min time t#1000ms; t#1000ms *)
	Start_Drucken_2__entry(P1);
	Start_Drucken_2__action(N);
	Start_Drucken_2__exit(P0);
END_STEP
TRANSITION FROM Start_Drucken_2_ TO busy2_ := TRUE;
END_TRANSITION
STEP busy2_:
END_STEP
TRANSITION FROM busy2_ TO Done2_ := Drucker_busy;
END_TRANSITION
TRANSITION FROM busy2_ TO Msg_Printer2_ := not_busy;
END_TRANSITION
STEP Msg_Printer2_:
	Msg_Printer2__entry(P1);
	Msg_Printer2__action(N);
	Msg_Printer2__exit(P0);
END_STEP
TRANSITION FROM Msg_Printer2_ TO Set_Auto_Stop2_ := MsgOK;
END_TRANSITION
STEP Set_Auto_Stop2_:
	Set_Auto_Stop2__action(N);
END_STEP
TRANSITION FROM Set_Auto_Stop2_ TO SeqEnd := AutoStop;
END_TRANSITION
STEP Done2_:
END_STEP
TRANSITION FROM Done2_ TO Kamera_aktiv_2_ := Drucker_fertig;
END_TRANSITION
STEP Kamera_aktiv_2_:
	Kamera_aktiv_2__exit(P0);
END_STEP
TRANSITION FROM Kamera_aktiv_2_ TO Start_Kamera_2_ := aktiv;
END_TRANSITION
TRANSITION FROM Kamera_aktiv_2_ TO Print_OK_2_ := TRUE;
END_TRANSITION
STEP Start_Kamera_2_:
	Start_Kamera_2__action(N);
END_STEP
TRANSITION FROM Start_Kamera_2_ TO Step71 := Busy;
END_TRANSITION
STEP Step71:
	Step71_entry(P1);
END_STEP
TRANSITION FROM Step71 TO Verarbeitet_Bild_2_ := Done;
END_TRANSITION
TRANSITION FROM Step71 TO Print_OK_2_ := CamNotAktiv;
END_TRANSITION
TRANSITION FROM Step71 TO Start_Kamera_2_ := CamDone;
END_TRANSITION
STEP Verarbeitet_Bild_2_:
	Verarbeitet_Bild_2__entry(P1);
END_STEP
TRANSITION FROM Verarbeitet_Bild_2_ TO Schwenken_2_90_Grad := TRUE;
END_TRANSITION
STEP Print_OK_2_:
	Print_OK_2__exit(P0);
END_STEP
TRANSITION FROM Print_OK_2_ TO Schwenken_2_90_Grad := TRUE;
END_TRANSITION
STEP Schwenken_2_90_Grad:
	Schwenken_2_90_Grad_entry(P1);
END_STEP
TRANSITION FROM Schwenken_2_90_Grad TO ResetNokCounter := StateOk;
END_TRANSITION
STEP CheckCounter:
	CheckCounter_entry(P1);
END_STEP
TRANSITION FROM CheckCounter TO CheckMode := CounterOK;
END_TRANSITION
TRANSITION FROM CheckCounter TO Msg_Cam := Nok_Cont;
END_TRANSITION
TRANSITION FROM CheckCounter TO Msg_Cam_Percent := Nok_Percent;
END_TRANSITION
TRANSITION FROM CheckCounter TO Step107 := Dummytest;
END_TRANSITION
STEP Msg_Cam:
	Msg_Cam_entry(P1);
	Msg_Cam_action(N);
	Msg_Cam_exit(P0);
END_STEP
TRANSITION FROM Msg_Cam TO Counter_Reset__ := MsgOK;
END_TRANSITION
STEP Counter_Reset__:
	Counter_Reset___entry(P1);
END_STEP
TRANSITION FROM Counter_Reset__ TO CheckMode := TRUE;
END_TRANSITION
STEP Step107:
END_STEP
TRANSITION FROM Step107 TO Step113 := Robo_free;
END_TRANSITION
STEP Step113:
END_STEP
TRANSITION FROM Step113 TO Drehen_links_0_Grad_ := 180_Grad_;
END_TRANSITION
TRANSITION FROM Step113 TO Drehen_rechts_180_Grad__ := 0_Grad_;
END_TRANSITION
STEP Drehen_links_0_Grad_:
	Drehen_links_0_Grad__entry(P1);
	Drehen_links_0_Grad__action(N);
	Drehen_links_0_Grad__exit(P0);
END_STEP
TRANSITION FROM Drehen_links_0_Grad_ TO DummyTestEnd := StateOk;
END_TRANSITION
STEP Drehen_rechts_180_Grad__:
	Drehen_rechts_180_Grad___entry(P1);
	Drehen_rechts_180_Grad___action(N);
	Drehen_rechts_180_Grad___exit(P0);
END_STEP
TRANSITION FROM Drehen_rechts_180_Grad__ TO DummyTestEnd := StateOk;
END_TRANSITION
STEP DummyTestEnd:
END_STEP
TRANSITION FROM DummyTestEnd TO SeqEnd := end;
END_TRANSITION
STEP Msg_Cam_Percent:
	Msg_Cam_Percent_entry(P1);
	Msg_Cam_Percent_action(N);
	Msg_Cam_Percent_exit(P0);
END_STEP
TRANSITION FROM Msg_Cam_Percent TO Counter_Reset__ := MsgOK;
END_TRANSITION
STEP CheckMode:
END_STEP
TRANSITION FROM CheckMode TO SeqEnd := AutoRun;
END_TRANSITION
TRANSITION FROM CheckMode TO JumpAutoStop_ := AutoStop;
END_TRANSITION
STEP JumpAutoStop_: (*  *)
	JumpAutoStop__action(N);
	JumpAutoStop__exit(P0);
END_STEP
TRANSITION FROM JumpAutoStop_ TO SeqEnd := StateOk;
END_TRANSITION
STEP SeqEnd: (* -> WAIT *)
	SeqEnd_action(N);
END_STEP
TRANSITION FROM SeqEnd TO WaitForStart := TRUE;
END_TRANSITION

ACTION Init_action:
Start:=FALSE;
State:=STATE_WAIT;
MsgOK:=FALSE;
MsgCancel:=FALSE;
SFCRun:=FALSE;
Result:=RESULT_NON;
NokCounter:=0;
LoopCounter :=0;

ST02_S1_70K61_A1.SetSignalHigh	:= FALSE;
ST02_S1_70K61_A1.SetSignalLow	:= TRUE;
END_ACTION

ACTION Dummytest_not_End_entry:
MessageHandler.ClearMessageLines(sVisu:=Visu.Message);
END_ACTION

ACTION Dummytest_not_End_action:
MessageHandler.Msg.ID:='PM151';
MessageHandler.Msg.Name:='DummyTest';
MessageHandler.Msg.Text:=' Dummy Pruefung wurde nicht beende, Anlage leeräumen ';
MessageHandler.Msg.Color:=Color.yellow;
MessageHandler.Msg.Station:=1;


MessageHandler(
	Prio:=2, 								(*1=highest, .. , 4=lowest*)
	Btn1Addr:=ADR(MsgOk),						(*Address of Button1 , if Zero then Button is unvisible*)
	Btn2Addr:=0,						(*Address of Button2 , if Zero then Button is unvisible*)
	sVisu:=Visu.Message);
END_ACTION

ACTION Dummytest_not_End_exit:
MsgOk:=FALSE;
MsgCancel:=FALSE;

MP.ST02.DummyPruefung_93pol := FALSE;
END_ACTION

ACTION TDA_Luft_NOK_entry:
MessageHandler.ClearMessageLines(sVisu:=Visu.Message);
END_ACTION

ACTION TDA_Luft_NOK_action:
MessageHandler.Msg.ID:='PM150';
MessageHandler.Msg.Name:='TDA Druckschalter';
MessageHandler.Msg.Text:='ST02 Druckschalter Wartungseinheit Hauptluft min.6 bar';
MessageHandler.Msg.Color:=Color.red;
MessageHandler.Msg.Station:=1;


MessageHandler(
	Prio:=2, 							(*1=highest, .. , 4=lowest*)
	Btn1Addr:=ADR(MsgOk),			(*Address of Button1 , if Zero then Button is unvisible*)
	Btn2Addr:=,						(*Address of Button2 , if Zero then Button is unvisible*)
	sVisu:=Visu.Message);
END_ACTION

ACTION TDA_Luft_NOK_exit:
MsgOk:=FALSE;
MsgCancel:=FALSE;
END_ACTION

ACTION WaitForStart_entry:
turn_done:=FALSE;
END_ACTION

ACTION WaitForStart_action:
IF 	Start   THEN
	State:=STATE_RUN;
	Result:=RESULT_NON;
	SFCTimeStart:=TIME();
	Start:=FALSE;
(*ELSE*)
ELSE
	State:=STATE_WAIT;
	MsgOK:=FALSE;
	MsgCancel:=FALSE;
	SFCRun:=FALSE;
END_IF
END_ACTION

ACTION Kamera_nicht_bb_entry:
MessageHandler.ClearMessageLines(sVisu:=Visu.Message);
END_ACTION

ACTION Kamera_nicht_bb_action:
MessageHandler.Msg.ID:='PM152';
MessageHandler.Msg.Name:='Check Camera';
MessageHandler.Msg.Text:='Sesopart Kamera ist nicht betriebsbereit';
MessageHandler.Msg.Color:=Color.red;
MessageHandler.Msg.Station:=1;


MessageHandler(
	Prio:=2, 						(*1=highest, .. , 4=lowest*)
	Btn1Addr:=ADR(MsgOk),			(*Address of Button1 , if Zero then Button is unvisible*)
	Btn2Addr:=,						(*Address of Button2 , if Zero then Button is unvisible*)
	sVisu:=Visu.Message);
END_ACTION

ACTION Kamera_nicht_bb_exit:
MsgOk:=FALSE;
MsgCancel:=FALSE;
ST02_DT_95_A1.b_quitt:=TRUE;
END_ACTION

ACTION Drucker_nicht_bb_entry:
MessageHandler.ClearMessageLines(sVisu:=Visu.Message);
END_ACTION

ACTION Drucker_nicht_bb_action:
MessageHandler.Msg.ID:='PM158';
MessageHandler.Msg.Name:='Check Drucker';
MessageHandler.Msg.Text:='Tampondrucker ist nicht betriebsbereit';
MessageHandler.Msg.Color:=Color.red;
MessageHandler.Msg.Station:=1;


MessageHandler(
	Prio:=2, 							(*1=highest, .. , 4=lowest*)
	Btn1Addr:=ADR(MsgOk),			(*Address of Button1 , if Zero then Button is unvisible*)
	Btn2Addr:=,						(*Address of Button2 , if Zero then Button is unvisible*)
	sVisu:=Visu.Message);
END_ACTION

ACTION Drucker_nicht_bb_exit:
MsgOk:=FALSE;
MsgCancel:=FALSE;
ST02_DT_95_A1.b_quitt:=TRUE;
END_ACTION

ACTION Drehen_links_0_Grad_entry:
MP.ST02.TableData:=PushData(MP.ST02.TableData);
END_ACTION

ACTION Drehen_links_0_Grad_action:
ST02_62_Y6.MoveInit:=TRUE;
END_ACTION

ACTION Drehen_links_0_Grad_exit:
turn_done:=TRUE;
END_ACTION

ACTION setPartState_entry:
MP.ST02.TableData[2].ProcessData.	Result:=99;	(*   0 = Teil noch nicht bearbeitet bzw. Nest leer*)
											(*   1 =  Oberseite OK*)
											(*  11 = Oberseite und Unterseite OK*)
											(*  99 = Teil ist NOK	*)
END_ACTION

ACTION Schwenken_1_180_Grad_entry:
(*auf 0 Grad*)
ST02_Schwenkarm[1].b_180_grad:=TRUE;
END_ACTION

ACTION Fixieren_1_close_action:
ST02_62_Y17.MoveWork:=TRUE;
END_ACTION

ACTION Start_Drucken_1_entry:
ST02_S1_70K61_A1.SetSignalHigh	:= FALSE;
ST02_S1_70K61_A1.SetSignalLow	:= TRUE;
END_ACTION

ACTION Start_Drucken_1_action:
ST02_S1_70K61_A1.SetSignalHigh	:= TRUE;
ST02_S1_70K61_A1.SetSignalLow	:= FALSE;
END_ACTION

ACTION Start_Drucken_1_exit:
ST02_S1_70K61_A1.SetSignalHigh	:= FALSE;
ST02_S1_70K61_A1.SetSignalLow	:= TRUE;
END_ACTION

ACTION Msg_Printer_entry:
MessageHandler.ClearMessageLines(sVisu:=Visu.Message);
END_ACTION

ACTION Msg_Printer_action:
MessageHandler.Msg.ID:='PM153';
MessageHandler.Msg.Name:='Error Printer';
MessageHandler.Msg.Text:='keine Rückmeldung vom Tampondrucker!';

MessageHandler.Msg.Color:=Color.red;
MessageHandler.Msg.Station:=3;

MessageHandler(
	Prio:=2, 								(*1=highest, .. , 4=lowest*)
	Btn1Addr:=ADR(MsgOk),				(*Address of Button1 , if Zero then Button is unvisible*)
	Btn2Addr:=0(*ADR(MsgCancel)*),			(*Address of Button2 , if Zero then Button is unvisible*)
	sVisu:=Visu.Message);
END_ACTION

ACTION Msg_Printer_exit:
MsgOk:=FALSE;
MsgCancel:=FALSE;
END_ACTION

ACTION Set_Auto_Stop_action:
ModeSelect.AskForAutoStop:=TRUE;
END_ACTION

ACTION Kamera_aktiv_1_exit:
RepeatCounter:=0;
END_ACTION

ACTION Start_Kamera_1_action:
IF NOT MP.ST02.SensopartEthernet THEN
	ST02_DT_95_A1.i16_job := TD.Sensopart_CamProgNo +1;		 (*Kamera Farberkennung*)
	ST02_DT_95_A1.b_start := TRUE;
ELSE
	ST02_DT_95_A2.JobNo := TD.Sensopart_CamProgNo +1;
	ST02_DT_95_A2.st_ctrl_in.b_start := TRUE;
END_IF
END_ACTION

ACTION Step69_entry:
IF NOT MP.ST02.SensopartEthernet THEN
	ST02_DT_95_A1.b_start := FALSE;	 (*Kamera Farberkennung*)
ELSE
	ST02_DT_95_A2.st_ctrl_in.b_start := FALSE;
END_IF

RepeatCounter:=RepeatCounter+1;
END_ACTION

ACTION Verarbeitet_Bild_1_entry:
(*Erkläfung der Auswertung:
In der Produktion wird  nur OK und NOK ausgwertet:
   0 = Teil noch nicht bearbeitet bzw. Nest leer
   1 =  Druck ist OK
   9 = Druck ist NOK
Bei der Dummyprüfung muss passend zum Dummy rot, blau oder beide NOK sein:
   6= Teil roter und blauer Druck NOK ist nur bei der Dummyprüfung aktiv
   7= Teil roter Druck NOKist nur bei der Dummyprüfung aktiv
   8= Teil blauer Druck NOK ist nur bei der Dummyprüfung aktiv
*)

(*Produktion Ansteuerung Sensopart über Ethernet*)
IF MP.ST02.SensopartEthernet  AND NOT MP.ST02.DummyPruefung_93pol THEN
	IF MP.ST02.CamOn THEN
			IF 	ST02_DT_95_A2.b_Kam_Pruef_IO AND	 (*Kamera Farberkennung*)
				NOT ST02_DT_95_A2.b_Kam_Pruef_NIO THEN
				MP.ST02.TableData[2].ProcessData.Result:=MP.ST02.TableData[2].ProcessData.Result:=1;
			ELSE
				MP.ST02.TableData[2].ProcessData.Result:=MP.ST02.TableData[2].ProcessData.Result:=9;
			END_IF
	ELSE
			MP.ST02.TableData[2].ProcessData.Result:=11;	(*   0 = Teil noch nicht bearbeitet bzw. Nest leer*)
	END_IF

(*Produktion Ansteuerung Sensopart über digitale Ein- und Ausgänge*)
ELSIF NOT MP.ST02.SensopartEthernet AND NOT MP.ST02.DummyPruefung_93pol  THEN
		IF MP.ST02.CamOn THEN
	
			IF 	ST02_DT_95_A1.Ergebnis_IO AND	 (*Kamera Farberkennung*)
				NOT ST02_DT_95_A1.Ergebnis_NIO THEN
				MP.ST02.TableData[2].ProcessData.Result:=MP.ST02.TableData[2].ProcessData.Result:=1;
			ELSE

				MP.ST02.TableData[2].ProcessData.Result:=MP.ST02.TableData[2].ProcessData.Result:=9;
			END_IF
		ELSE
			MP.ST02.TableData[2].ProcessData.Result:=11;	(*   0 = Teil noch nicht bearbeitet bzw. Nest leer*)
		END_IF

(*Dummyprüfung Auswertung ist nur über Ehternet möglich*)
ELSIF MP.ST02.SensopartEthernet  AND MP.ST02.DummyPruefung_93pol THEN
	IF MP.ST02.CamOn THEN
			IF 	ST02_DT_95_A2.b_Kam_Pruef_IO AND	 (*Kamera Farberkennung*)
				NOT ST02_DT_95_A2.b_Kam_Pruef_NIO THEN
			MP.ST02.TableData[2].ProcessData.Result:=MP.ST02.TableData[2].ProcessData.Result:=1;
		(*roter Druck schlecht*)
			ELSIF ST02_DT_95_A2.RecvDataString = CONCAT('5FFPFP', INT_TO_STRING(ST02_DT_95_A2.JobNo)) THEN
				MP.ST02.TableData[2].ProcessData.Result:=MP.ST02.TableData[2].ProcessData.Result:=7;
		(*blauer Druck schlecht*)
			ELSIF ST02_DT_95_A2.RecvDataString = CONCAT('5FFPPF', INT_TO_STRING(ST02_DT_95_A2.JobNo)) THEN
				MP.ST02.TableData[2].ProcessData.Result:=MP.ST02.TableData[2].ProcessData.Result:=8;
		(*beide Druck schlecht*)
			ELSIF ST02_DT_95_A2.RecvDataString = CONCAT('5FFPFF', INT_TO_STRING(ST02_DT_95_A2.JobNo)) THEN
				MP.ST02.TableData[2].ProcessData.Result:=MP.ST02.TableData[2].ProcessData.Result:=6;

			ELSE
				MP.ST02.TableData[2].ProcessData.Result:=MP.ST02.TableData[2].ProcessData.Result:=9;

			END_IF
	END_IF
END_IF

RepeatCounter:=RepeatCounter+1;
END_ACTION

ACTION Print_OK_1_exit:
MP.ST02.TableData[2].ProcessData.Result:=1;	(*   0 = Teil noch nicht bearbeitet bzw. Nest leer*)
											(*   1 =  Oberseite OK*)
											(*  11 = Oberseite und Unterseite OK*)
											(*  99 = Teil ist NOK	*)
END_ACTION

ACTION Fixieren_1_open_action:
ST02_62_Y17.MoveInit:=TRUE;
END_ACTION

ACTION Schwenken_1_0_Grad_entry:
(*auf 180 Grad*)
ST02_Schwenkarm[1].b_0_grad:=TRUE;
END_ACTION

ACTION Start_Drucken_2_entry:
ST02_S1_70K61_A1.SetSignalHigh	:= FALSE;
ST02_S1_70K61_A1.SetSignalLow	:= TRUE;
END_ACTION

ACTION Start_Drucken_2_action:
ST02_S1_70K61_A1.SetSignalHigh	:= TRUE;
ST02_S1_70K61_A1.SetSignalLow	:= FALSE;
END_ACTION

ACTION Start_Drucken_2_exit:
ST02_S1_70K61_A1.SetSignalHigh	:= FALSE;
ST02_S1_70K61_A1.SetSignalLow	:= TRUE;
END_ACTION

ACTION Msg_Printer2_entry:
MessageHandler.ClearMessageLines(sVisu:=Visu.Message);
END_ACTION

ACTION Msg_Printer2_action:
MessageHandler.Msg.Name:='Error Printer';

MessageHandler.Msg.Text:='keine Rückmeldung vom Tampondrucker!';

MessageHandler.Msg.Color:=Color.red;
MessageHandler.Msg.Station:=3;

MessageHandler(
	Prio:=2, 								(*1=highest, .. , 4=lowest*)
	Btn1Addr:=ADR(MsgOk),				(*Address of Button1 , if Zero then Button is unvisible*)
	Btn2Addr:=0(*ADR(MsgCancel)*),			(*Address of Button2 , if Zero then Button is unvisible*)
	sVisu:=Visu.Message);
END_ACTION

ACTION Msg_Printer2_exit:
MsgOk:=FALSE;
MsgCancel:=FALSE;
END_ACTION

ACTION Set_Auto_Stop2_action:
ModeSelect.AskForAutoStop:=TRUE;
END_ACTION

ACTION Kamera_aktiv_2_exit:
RepeatCounter:=0;
END_ACTION

ACTION Start_Kamera_2_action:
IF NOT MP.ST02.SensopartEthernet THEN
ST02_DT_95_A1.i16_job := TD.Sensopart_CamProgNo;	 (*Kamera Farberkennung*)
ST02_DT_95_A1.b_start := TRUE;
ELSE
	ST02_DT_95_A2.JobNo := TD.Sensopart_CamProgNo;
	ST02_DT_95_A2.st_ctrl_in.b_start := TRUE;
END_IF
END_ACTION

ACTION Step72_entry:
IF NOT MP.ST02.SensopartEthernet THEN
ST02_DT_95_A1.b_start := FALSE;	 (*Kamera Farberkennung*)
RepeatCounter:=RepeatCounter+1;
ELSE
	ST02_DT_95_A2.st_ctrl_in.b_start := FALSE;
	RepeatCounter:=RepeatCounter+1;
END_IF
END_ACTION

ACTION Verarbeitet_Bild_2_entry:
(*Erkläfung der Auswertung:
In der Produktion wird  nur OK und NOK ausgwertet:
   0 = Teil noch nicht bearbeitet bzw. Nest leer
   1 =  Druck ist OK
   9 = Druck ist NOK
Bei der Dummyprüfung muss passend zum Dummy rot, blau oder beide NOK sein:
   6= Teil roter und blauer Druck NOK ist nur bei der Dummyprüfung aktiv
   7= Teil roter Druck NOKist nur bei der Dummyprüfung aktiv
   8= Teil blauer Druck NOK ist nur bei der Dummyprüfung aktiv
*)

(*Produktion Ansteuerung Sensopart über Ethernet*)
IF MP.ST02.SensopartEthernet  AND NOT MP.ST02.DummyPruefung_93pol THEN
	IF MP.ST02.CamOn THEN
			IF 	ST02_DT_95_A2.b_Kam_Pruef_IO AND	 (*Kamera Farberkennung*)
				NOT ST02_DT_95_A2.b_Kam_Pruef_NIO THEN
				MP.ST02.TableData[2].ProcessData.Result:=MP.ST02.TableData[2].ProcessData.Result+10;
			ELSE
				MP.ST02.TableData[2].ProcessData.Result:=MP.ST02.TableData[2].ProcessData.Result+90;
			END_IF
	ELSE
			MP.ST02.TableData[2].ProcessData.Result:=11;	(*   0 = Teil noch nicht bearbeitet bzw. Nest leer*)
	END_IF

(*Produktion Ansteuerung Sensopart über digitale Ein- und Ausgänge*)
ELSIF NOT MP.ST02.SensopartEthernet AND NOT MP.ST02.DummyPruefung_93pol  THEN
		IF MP.ST02.CamOn THEN
			IF 	ST02_DT_95_A1.Ergebnis_IO AND	 (*Kamera Farberkennung*)
				NOT ST02_DT_95_A1.Ergebnis_NIO THEN
				MP.ST02.TableData[2].ProcessData.Result:=MP.ST02.TableData[2].ProcessData.Result+10;
			ELSE
				MP.ST02.TableData[2].ProcessData.Result:=MP.ST02.TableData[2].ProcessData.Result+90;
			END_IF
		ELSE
			MP.ST02.TableData[2].ProcessData.Result:=11;	(*   0 = Teil noch nicht bearbeitet bzw. Nest leer*)
		END_IF

(*Dummyprüfung Auswertung ist nur über Ehternet möglich*)
ELSIF MP.ST02.SensopartEthernet  AND MP.ST02.DummyPruefung_93pol THEN
	IF MP.ST02.CamOn THEN
			IF 	ST02_DT_95_A2.b_Kam_Pruef_IO AND	 (*Kamera Farberkennung*)
				NOT ST02_DT_95_A2.b_Kam_Pruef_NIO THEN
			MP.ST02.TableData[2].ProcessData.Result:=MP.ST02.TableData[2].ProcessData.Result+10;
		(*roter Druck schlecht*)
			ELSIF ST02_DT_95_A2.RecvDataString = CONCAT('5FFPFP', INT_TO_STRING(ST02_DT_95_A2.JobNo)) THEN
				MP.ST02.TableData[2].ProcessData.Result:=MP.ST02.TableData[2].ProcessData.Result+70;
		(*blauer Druck schlecht*)
			ELSIF ST02_DT_95_A2.RecvDataString = CONCAT('5FFPPF', INT_TO_STRING(ST02_DT_95_A2.JobNo)) THEN
				MP.ST02.TableData[2].ProcessData.Result:=MP.ST02.TableData[2].ProcessData.Result+80;
		(*beide Druck schlecht*)
			ELSIF ST02_DT_95_A2.RecvDataString = CONCAT('5FFPFF', INT_TO_STRING(ST02_DT_95_A2.JobNo)) THEN
				MP.ST02.TableData[2].ProcessData.Result:=MP.ST02.TableData[2].ProcessData.Result+60;

			ELSE
				MP.ST02.TableData[2].ProcessData.Result:=MP.ST02.TableData[2].ProcessData.Result+90;

			END_IF
	END_IF
END_IF
END_ACTION

ACTION Print_OK_1__exit:
MP.ST02.TableData[2].ProcessData.Result:=MP.ST02.TableData[2].ProcessData.Result +10;	(*   0 = Teil noch nicht bearbeitet bzw. Nest leer*)
											(*   1 =  Oberseite OK*)
											(*  11 = Oberseite und Unterseite OK*)
											(*  99 = Teil ist NOK	*)
END_ACTION

ACTION Schwenken_1_90_Grad_entry:
(*auf 90 Grad*)
ST02_Schwenkarm[1].b_90_grad:=TRUE;
END_ACTION

ACTION ResetNokCounter_entry:
(*Register um eins nach hinten schieben*)
i:=0;
FOR i:=100 TO 2 BY-1 DO
   NokPercent[i] := NokPercent[i-1];
END_FOR

IF	MP.ST02.TableData[2].ProcessData.Result = 11 THEN
	NokCounter:=0;
	NokPercent[1] := FALSE;
ELSIF NOT MP.ST02.DummyPruefung_93pol THEN
	gNokPartsColorCam := gNokPartsColorCam+1;
	NokCounter:=NokCounter+1;
	NokPercent[1] := TRUE;
END_IF

(*Ergebnise in Puffer eintragen für Dummyprüfung*)
i:=0;
FOR i:=10 TO 2 BY-1 DO
	ResultBuffer[i]:=ResultBuffer[i-1];
END_FOR
ResultBuffer[1]:=MP.ST02.TableData[2].ProcessData.Result;
END_ACTION

ACTION Drehen_rechts_180_Grad_entry:
MP.ST02.TableData:=PushData(MP.ST02.TableData);
END_ACTION

ACTION Drehen_rechts_180_Grad_action:
ST02_62_Y6.MoveWork:=TRUE;
END_ACTION

ACTION Drehen_rechts_180_Grad_exit:
turn_done:=TRUE;
END_ACTION

ACTION setPartState__entry:
MP.ST02.TableData[2].ProcessData.	Result:=99;	(*   0 = Teil noch nicht bearbeitet bzw. Nest leer*)
											(*   1 =  Oberseite OK*)
											(*  11 = Oberseite und Unterseite OK*)
											(*  99 = Teil ist NOK	*)
END_ACTION

ACTION Schwenken_2_180_Grad_entry:
(*auf 0 Grad*)
ST02_Schwenkarm[2].b_180_grad:=TRUE;
END_ACTION

ACTION Fixieren_2_close_action:
ST02_62_Y18.MoveWork:=TRUE;
END_ACTION

ACTION Start_Drucken_1__entry:
ST02_S1_70K61_A1.SetSignalHigh	:= FALSE;
ST02_S1_70K61_A1.SetSignalLow	:= TRUE;
END_ACTION

ACTION Start_Drucken_1__action:
ST02_S1_70K61_A1.SetSignalHigh	:= TRUE;
ST02_S1_70K61_A1.SetSignalLow	:= FALSE;
END_ACTION

ACTION Start_Drucken_1__exit:
ST02_S1_70K61_A1.SetSignalHigh	:= FALSE;
ST02_S1_70K61_A1.SetSignalLow	:= TRUE;
END_ACTION

ACTION Msg_Printer__entry:
MessageHandler.ClearMessageLines(sVisu:=Visu.Message);
END_ACTION

ACTION Msg_Printer__action:
MessageHandler.Msg.ID:='PM153';
MessageHandler.Msg.Name:='Error Printer';
MessageHandler.Msg.Text:='keine Rückmeldung vom Tampondrucker!';
MessageHandler.Msg.Color:=Color.red;
MessageHandler.Msg.Station:=3;

MessageHandler(
	Prio:=2, 								(*1=highest, .. , 4=lowest*)
	Btn1Addr:=ADR(MsgOk),				(*Address of Button1 , if Zero then Button is unvisible*)
	Btn2Addr:=0(*ADR(MsgCancel)*),			(*Address of Button2 , if Zero then Button is unvisible*)
	sVisu:=Visu.Message);
END_ACTION

ACTION Msg_Printer__exit:
MsgOk:=FALSE;
MsgCancel:=FALSE;
END_ACTION

ACTION Set_AutoStop__action:
ModeSelect.AskForAutoStop:=TRUE;
END_ACTION

ACTION Kamera_aktiv_1__exit:
RepeatCounter:=0;
END_ACTION

ACTION Start_Kamera_1__action:
IF NOT MP.ST02.SensopartEthernet  THEN
	ST02_DT_95_A1.i16_job := TD.Sensopart_CamProgNo +1;	 (*Kamera Farberkennung*)
	ST02_DT_95_A1.b_start := TRUE;
ELSE
	ST02_DT_95_A2.JobNo := TD.Sensopart_CamProgNo +1;
	ST02_DT_95_A2.st_ctrl_in.b_start := TRUE;
END_IF
END_ACTION

ACTION Step70_entry:
IF NOT MP.ST02.SensopartEthernet  THEN
	ST02_DT_95_A1.b_start := FALSE;	 (*Kamera Farberkennung*)
ELSE
	ST02_DT_95_A2.st_ctrl_in.b_start := FALSE;
END_IF

RepeatCounter:=RepeatCounter+1;
END_ACTION

ACTION Verarbeitet_Bild_1__entry:
(*Erkläfung der Auswertung:
In der Produktion wird  nur OK und NOK ausgwertet:
   0 = Teil noch nicht bearbeitet bzw. Nest leer
   1 =  Druck ist OK
   9 = Druck ist NOK
Bei der Dummyprüfung muss passend zum Dummy rot, blau oder beide NOK sein:
   6= Teil roter und blauer Druck NOK ist nur bei der Dummyprüfung aktiv
   7= Teil roter Druck NOKist nur bei der Dummyprüfung aktiv
   8= Teil blauer Druck NOK ist nur bei der Dummyprüfung aktiv
*)


(*Produktion Ansteuerung Sensopart über Ethernet*)
IF MP.ST02.SensopartEthernet  AND NOT MP.ST02.DummyPruefung_93pol THEN
	IF MP.ST02.CamOn THEN
			IF 	ST02_DT_95_A2.b_Kam_Pruef_IO AND	 (*Kamera Farberkennung*)
				NOT ST02_DT_95_A2.b_Kam_Pruef_NIO THEN
				MP.ST02.TableData[2].ProcessData.Result:=MP.ST02.TableData[2].ProcessData.Result:=1;
			ELSE
				MP.ST02.TableData[2].ProcessData.Result:=MP.ST02.TableData[2].ProcessData.Result:=9;
			END_IF
	ELSE
			MP.ST02.TableData[2].ProcessData.Result:=11;	(*   0 = Teil noch nicht bearbeitet bzw. Nest leer*)
	END_IF

(*Produktion Ansteuerung Sensopart über digitale Ein- und Ausgänge*)
ELSIF NOT MP.ST02.SensopartEthernet AND NOT MP.ST02.DummyPruefung_93pol  THEN
		IF MP.ST02.CamOn THEN
			IF 	ST02_DT_95_A1.Ergebnis_IO AND	 (*Kamera Farberkennung*)
				NOT ST02_DT_95_A1.Ergebnis_NIO THEN
				MP.ST02.TableData[2].ProcessData.Result:=MP.ST02.TableData[2].ProcessData.Result:=1;
			ELSE
				MP.ST02.TableData[2].ProcessData.Result:=MP.ST02.TableData[2].ProcessData.Result:=9;
			END_IF
		ELSE
				MP.ST02.TableData[2].ProcessData.Result:=11;	(*   0 = Teil noch nicht bearbeitet bzw. Nest leer*)
		END_IF

(*Dummyprüfung Auswertung ist nur über Ehternet möglich*)
ELSIF MP.ST02.SensopartEthernet  AND MP.ST02.DummyPruefung_93pol THEN
	IF MP.ST02.CamOn THEN
			IF 	ST02_DT_95_A2.b_Kam_Pruef_IO AND	 (*Kamera Farberkennung*)
				NOT ST02_DT_95_A2.b_Kam_Pruef_NIO THEN
				MP.ST02.TableData[2].ProcessData.Result:=MP.ST02.TableData[2].ProcessData.Result:=1;
		(*roter Druck schlecht*)
			ELSIF ST02_DT_95_A2.RecvDataString = CONCAT('5FFPFP', INT_TO_STRING(ST02_DT_95_A2.JobNo)) THEN
				MP.ST02.TableData[2].ProcessData.Result:=MP.ST02.TableData[2].ProcessData.Result:=7;
		(*blauer Druck schlecht*)
			ELSIF ST02_DT_95_A2.RecvDataString = CONCAT('5FFPPF', INT_TO_STRING(ST02_DT_95_A2.JobNo)) THEN
				MP.ST02.TableData[2].ProcessData.Result:=MP.ST02.TableData[2].ProcessData.Result:=8;
		(*beide Druck schlecht*)
				ELSIF ST02_DT_95_A2.RecvDataString = CONCAT('5FFPFF', INT_TO_STRING(ST02_DT_95_A2.JobNo)) THEN
				MP.ST02.TableData[2].ProcessData.Result:=MP.ST02.TableData[2].ProcessData.Result:=6;

			ELSE
				MP.ST02.TableData[2].ProcessData.Result:=MP.ST02.TableData[2].ProcessData.Result:=9;

			END_IF
	END_IF
END_IF

RepeatCounter:=RepeatCounter+1;
END_ACTION

ACTION Print_OK_2_exit:
MP.ST02.TableData[2].ProcessData.Result:=1;	(*   0 = Teil noch nicht bearbeitet bzw. Nest leer*)
											(*   1 =  Oberseite OK*)
											(*  11 = Oberseite und Unterseite OK*)
											(*  99 = Teil ist NOK	*)
END_ACTION

ACTION Fixieren_2_open_action:
ST02_62_Y18.MoveInit:=TRUE;
END_ACTION

ACTION Schwenken_2_0_Grad_entry:
(*auf 180 Grad*)
ST02_Schwenkarm[2].b_0_grad:=TRUE;
END_ACTION

ACTION Start_Drucken_2__entry:
ST02_S1_70K61_A1.SetSignalHigh	:= FALSE;
ST02_S1_70K61_A1.SetSignalLow	:= TRUE;
END_ACTION

ACTION Start_Drucken_2__action:
ST02_S1_70K61_A1.SetSignalHigh	:= TRUE;
ST02_S1_70K61_A1.SetSignalLow	:= FALSE;
END_ACTION

ACTION Start_Drucken_2__exit:
ST02_S1_70K61_A1.SetSignalHigh	:= FALSE;
ST02_S1_70K61_A1.SetSignalLow	:= TRUE;
END_ACTION

ACTION Msg_Printer2__entry:
MessageHandler.ClearMessageLines(sVisu:=Visu.Message);
END_ACTION

ACTION Msg_Printer2__action:
MessageHandler.Msg.ID:='PM153';
MessageHandler.Msg.Name:='Error Printer';
MessageHandler.Msg.Text:='keine Rückmeldung vom Tampondrucker!';
MessageHandler.Msg.Color:=Color.red;
MessageHandler.Msg.Station:=3;

MessageHandler(
	Prio:=2, 								(*1=highest, .. , 4=lowest*)
	Btn1Addr:=ADR(MsgOk),				(*Address of Button1 , if Zero then Button is unvisible*)
	Btn2Addr:=0(*ADR(MsgCancel)*),			(*Address of Button2 , if Zero then Button is unvisible*)
	sVisu:=Visu.Message);
END_ACTION

ACTION Msg_Printer2__exit:
MsgOk:=FALSE;
MsgCancel:=FALSE;
END_ACTION

ACTION Set_Auto_Stop2__action:
ModeSelect.AskForAutoStop:=TRUE;
END_ACTION

ACTION Kamera_aktiv_2__exit:
RepeatCounter:=0;
END_ACTION

ACTION Start_Kamera_2__action:
IF NOT MP.ST02.SensopartEthernet  THEN
	ST02_DT_95_A1.i16_job := TD.Sensopart_CamProgNo;	 (*Kamera Farberkennung*)
	ST02_DT_95_A1.b_start := TRUE;
ELSE
	ST02_DT_95_A2.JobNo := TD.Sensopart_CamProgNo;
	ST02_DT_95_A2.st_ctrl_in.b_start := TRUE;
END_IF
END_ACTION

ACTION Step71_entry:
IF NOT MP.ST02.SensopartEthernet  THEN
	ST02_DT_95_A1.b_start := FALSE;	 (*Kamera Farberkennung*)
	RepeatCounter:=RepeatCounter+1;
ELSE
	ST02_DT_95_A2.st_ctrl_in.b_start := FALSE;
	RepeatCounter:=RepeatCounter+1;
END_IF
END_ACTION

ACTION Verarbeitet_Bild_2__entry:
(*Erkläfung der Auswertung:
In der Produktion wird  nur OK und NOK ausgwertet:
   0 = Teil noch nicht bearbeitet bzw. Nest leer
   1 =  Druck ist OK
   9 = Druck ist NOK
Bei der Dummyprüfung muss passend zum Dummy rot, blau oder beide NOK sein:
   6= Teil roter und blauer Druck NOK ist nur bei der Dummyprüfung aktiv
   7= Teil roter Druck NOKist nur bei der Dummyprüfung aktiv
   8= Teil blauer Druck NOK ist nur bei der Dummyprüfung aktiv
*)

(*Produktion Ansteuerung Sensopart über Ethernet*)
IF MP.ST02.SensopartEthernet AND NOT MP.ST02.DummyPruefung_93pol THEN
	IF MP.ST02.CamOn THEN
			IF 	ST02_DT_95_A2.b_Kam_Pruef_IO AND	 (*Kamera Farberkennung*)
				NOT ST02_DT_95_A2.b_Kam_Pruef_NIO THEN
				MP.ST02.TableData[2].ProcessData.Result:=MP.ST02.TableData[2].ProcessData.Result+10;
			ELSE
				MP.ST02.TableData[2].ProcessData.Result:=MP.ST02.TableData[2].ProcessData.Result+90;
			END_IF
	ELSE
				MP.ST02.TableData[2].ProcessData.Result:=11;	(*   0 = Teil noch nicht bearbeitet bzw. Nest leer*)
	END_IF

(*Produktion Ansteuerung Sensopart über digitale Ein- und Ausgänge*)
ELSIF NOT MP.ST02.SensopartEthernet  AND NOT MP.ST02.DummyPruefung_93pol  THEN
		IF MP.ST02.CamOn THEN
			IF 	ST02_DT_95_A1.Ergebnis_IO AND	 (*Kamera Farberkennung*)
				NOT ST02_DT_95_A1.Ergebnis_NIO THEN
				MP.ST02.TableData[2].ProcessData.Result:=MP.ST02.TableData[2].ProcessData.Result+10;
			ELSE
				MP.ST02.TableData[2].ProcessData.Result:=MP.ST02.TableData[2].ProcessData.Result+90;
			END_IF
		ELSE
				MP.ST02.TableData[2].ProcessData.Result:=11;	(*   0 = Teil noch nicht bearbeitet bzw. Nest leer*)
		END_IF

(*Dummyprüfung Auswertung ist nur über Ehternet möglich*)
ELSIF MP.ST02.SensopartEthernet AND MP.ST02.DummyPruefung_93pol THEN
	IF MP.ST02.CamOn THEN
			IF 	ST02_DT_95_A2.b_Kam_Pruef_IO AND	 (*Kamera Farberkennung*)
				NOT ST02_DT_95_A2.b_Kam_Pruef_NIO THEN
				MP.ST02.TableData[2].ProcessData.Result:=MP.ST02.TableData[2].ProcessData.Result+10;
		(*roter Druck schlecht*)
			ELSIF ST02_DT_95_A2.RecvDataString = CONCAT('5FFPFP', INT_TO_STRING(ST02_DT_95_A2.JobNo)) THEN
				MP.ST02.TableData[2].ProcessData.Result:=MP.ST02.TableData[2].ProcessData.Result+70;
		(*blauer Druck schlecht*)
			ELSIF ST02_DT_95_A2.RecvDataString = CONCAT('5FFPPF', INT_TO_STRING(ST02_DT_95_A2.JobNo)) THEN
				MP.ST02.TableData[2].ProcessData.Result:=MP.ST02.TableData[2].ProcessData.Result+80;
		(*beide Druck schlecht*)
			ELSIF ST02_DT_95_A2.RecvDataString = CONCAT('5FFPFF', INT_TO_STRING(ST02_DT_95_A2.JobNo)) THEN
				MP.ST02.TableData[2].ProcessData.Result:=MP.ST02.TableData[2].ProcessData.Result+60;

			ELSE
				MP.ST02.TableData[2].ProcessData.Result:=MP.ST02.TableData[2].ProcessData.Result+90;

			END_IF
	END_IF
END_IF


RepeatCounter:=RepeatCounter+1;
END_ACTION

ACTION Print_OK_2__exit:
MP.ST02.TableData[2].ProcessData.	Result:=MP.ST02.TableData[2].ProcessData.	Result +10;	(*   0 = Teil noch nicht bearbeitet bzw. Nest leer*)
											(*   1 =  Oberseite OK*)
											(*  11 = Oberseite und Unterseite OK*)
											(*  99 = Teil ist NOK	*)
END_ACTION

ACTION Schwenken_2_90_Grad_entry:
(*auf 180 Grad*)
ST02_Schwenkarm[2].b_90_grad:=TRUE;
END_ACTION

ACTION CheckCounter_entry:
(*Anzahl der Schlechtteile von den letzten 100 Prüfungen*)
IF NOT MP.ST02.DummyPruefung_93pol THEN
	i:=0;
	NokCounterPercent:=0;
	FOR i:=1 TO 100 BY 1 DO
  		IF	NokPercent[i] THEN
		NokCounterPercent:=NokCounterPercent+1;
		END_IF
	END_FOR
ELSE
	LoopCounter	:= LoopCounter +1;
END_IF
END_ACTION

ACTION Msg_Cam_entry:
MessageHandler.ClearMessageLines(sVisu:=Visu.Message);
END_ACTION

ACTION Msg_Cam_action:
MessageHandler.Msg.ID:='PM112';
MessageHandler.Msg.Name:='Sensopart Kam.-Erg. Prüfung  n.i.o:';
MessageHandler.Msg.Text:='Sensopart Kam.-Erg. Prüfung  n.i.o: Fehler in Folge';
MessageHandler.Msg.Color:=Color.red;
MessageHandler.Msg.Station:=3;
MessageHandler.MsgButton1Text:='continue';

MessageHandler(
	Prio:=2, 								(*1=highest, .. , 4=lowest*)
	Btn1Addr:=ADR(MsgOk),				(*Address of Button1 , if Zero then Button is unvisible*)
	Btn2Addr:=0(*ADR(MsgCancel)*),			(*Address of Button2 , if Zero then Button is unvisible*)
	sVisu:=Visu.Message);
END_ACTION

ACTION Msg_Cam_exit:
MsgOk:=FALSE;
MsgCancel:=FALSE;
END_ACTION

